	sErrorDescription1 := 'User High level error.  Illegal demand data was transmitted.';				
	sErrorDescription2 := 'Check program';				
					
9070:					
					
	sErrorDescription1 := 'User High level error.  Illegal demand data was transmitted.';				
	sErrorDescription2 := 'Check program';				
					
9071:					
					
	sErrorDescription1 := 'User High level error.  Illegal demand data was transmitted.';				
	sErrorDescription2 := 'Check program';				
					
9072:					
					
	sErrorDescription1 := 'User High level error.  Illegal demand data was transmitted.';				
	sErrorDescription2 := 'Check program';				
					
9073:					
					
	sErrorDescription1 := 'User High level error.  Illegal demand data was transmitted.';				
	sErrorDescription2 := 'Check program';				
					
9074:					
					
	sErrorDescription1 := 'User High level error.  Illegal demand data was transmitted.';				
	sErrorDescription2 := 'Check program';				
					
9075:					
					
	sErrorDescription1 := 'User High level error.  Illegal demand data was transmitted.';				
	sErrorDescription2 := 'Check program';				
					
9076:					
					
	sErrorDescription1 := 'User High level error.  Illegal demand data was transmitted.';				
	sErrorDescription2 := 'Check program';				
					
9077:					
					
	sErrorDescription1 := 'User High level error.  Illegal demand data was transmitted.';				
	sErrorDescription2 := 'Check program';				
					
9078:					
					
	sErrorDescription1 := 'User High level error.  Illegal demand data was transmitted.';				
	sErrorDescription2 := 'Check program';				
					
9079:					
					
	sErrorDescription1 := 'User High level error.  Illegal demand data was transmitted.';				
	sErrorDescription2 := 'Check program';				
					
9080:					
					
	sErrorDescription1 := 'User High level error.  Illegal demand data was transmitted.';				
	sErrorDescription2 := 'Check program';				
					
9081:					
					
	sErrorDescription1 := 'User High level error.  Illegal demand data was transmitted.';				
	sErrorDescription2 := 'Check program';				
					
9082:					
					
	sErrorDescription1 := 'User High level error.  Illegal demand data was transmitted.';				
	sErrorDescription2 := 'Check program';				
					
9083:					
					
	sErrorDescription1 := 'User High level error.  Illegal demand data was transmitted.';				
	sErrorDescription2 := 'Check program';				
					
9084:					
					
	sErrorDescription1 := 'User High level error.  Illegal demand data was transmitted.';				
	sErrorDescription2 := 'Check program';				
					
9085:					
					
	sErrorDescription1 := 'User High level error.  Illegal demand data was transmitted.';				
	sErrorDescription2 := 'Check program';				
					
9086:					
					
	sErrorDescription1 := 'User High level error.  Illegal demand data was transmitted.';				
	sErrorDescription2 := 'Check program';				
					
9087:					
					
	sErrorDescription1 := 'User High level error.  Illegal demand data was transmitted.';				
	sErrorDescription2 := 'Check program';				
					
9088:					
					
	sErrorDescription1 := 'User High level error.  Illegal demand data was transmitted.';				
	sErrorDescription2 := 'Check program';				
					
9089:					
					
	sErrorDescription1 := 'User High level error.  Illegal demand data was transmitted.';				
	sErrorDescription2 := 'Check program';				
					
9090:					
					
	sErrorDescription1 := 'User High level error.  Illegal demand data was transmitted.';				
	sErrorDescription2 := 'Check program';				
					
9091:					
					
	sErrorDescription1 := 'User High level error.  Illegal demand data was transmitted.';				
	sErrorDescription2 := 'Check program';				
					
9092:					
					
	sErrorDescription1 := 'User High level error.  Illegal demand data was transmitted.';				
	sErrorDescription2 := 'Check program';				
					
9093:					
					
	sErrorDescription1 := 'User High level error.  Illegal demand data was transmitted.';				
	sErrorDescription2 := 'Check program';				
					
9094:					
					
	sErrorDescription1 := 'User High level error.  Illegal demand data was transmitted.';				
	sErrorDescription2 := 'Check program';				
					
9095:					
					
	sErrorDescription1 := 'User High level error.  Illegal demand data was transmitted.';				
	sErrorDescription2 := 'Check program';				
					
9096:					
					
	sErrorDescription1 := 'User High level error.  Illegal demand data was transmitted.';				
	sErrorDescription2 := 'Check program';				
					
9097:					
					
	sErrorDescription1 := 'User High level error.  Illegal demand data was transmitted.';				
	sErrorDescription2 := 'Check program';				
					
9098:					
					
	sErrorDescription1 := 'User High level error.  Illegal demand data was transmitted.';				
	sErrorDescription2 := 'Check program';				
					
9099:					
					
	sErrorDescription1 := 'User High level error.  Illegal demand data was transmitted.';				
	sErrorDescription2 := 'Check program';				
		
		END_CASE
END_IF		
		
IF bErrorRCActive AND bLowLevelErrorRCActive  THEN
		
		CASE udiLowLevelErrorId OF
			

0030:	
	
	sErrorDescription1 := 'Hand error. LS release  Hand error signal is input';
	sErrorDescription2 := 'Restore with LS release operation';
	
0031:	
	
	sErrorDescription1 := 'Air pressure errorAir pressure error signal input';
	sErrorDescription2 := 'Check Air pressure';
	
0091:	
	
	sErrorDescription1 := 'Can not access the Special signThis signal cannot be used in duplicate';
	sErrorDescription2 := 'Change output No or special output assignment parameter';
	
0092:	
	
	sErrorDescription1 := ' Can not use Electric hand signaThe output signal for the electric hand cannot be used';
	sErrorDescription2 := 'Correct the program';
	
0095:	
	
	sErrorDescription1 := ' Brake release switch is turniCannot execute while brake release switch is turning on.';
	sErrorDescription2 := 'Please check the brake release switch and turn it off.';
	
0101:	
	
	sErrorDescription1 := 'Temperature in the Controlle FAN check or Filter at the bottom on Controller becomes old';
	sErrorDescription2 := 'Please exchange the filter to new filter or clean up the filter';
	
0104:	
	
	sErrorDescription1 := ' Temp. in robot CPU is too higAmbient temperature of robot CPU becomes high';
	sErrorDescription2 := 'Please lower ambient temperature to the specification range';
	
0110:	
	
	sErrorDescription1 := ' Overload(UPS)The UPS is spent';
	sErrorDescription2 := 'Replace the UPS';
	
0113:	
	
	sErrorDescription1 := ' UPS power supply error UPS power supply is out OF range';
	sErrorDescription2 := 'Check the UPS power supply';
	
0301:	
	
	sErrorDescription1 := ' CR800 test L-ErrorGeneral-purpose L-Error for the function test of CR800';
	sErrorDescription2 := 'Check the embedded message';
	
0480:	
	
	sErrorDescription1 := ' THR-RR error(Add.Axis)Overheating of the regenerative resistor (Add.Axis) was detected';
	sErrorDescription2 := 'Exchange the cooling fan of the regenerative resistor (Add.Axis)';
	
1640:	
	
	sErrorDescription1 := 'Cannot servo ON (DEADMAN OFF)The servo cannot be turned ON while the deadman switch OFF';
	sErrorDescription2 := 'Turn the deadman switch ON before turning the servo ON';
	
1820:	
	
	sErrorDescription1 := 'Pos. data disagree.Check origPosition data changed during power off';
	sErrorDescription2 := 'Check the origin, re-install if neccesary';
	
1830:	
	
	sErrorDescription1 := 'JRC. Exseeds the Pos. limitExceeds the pos. limit by JRC command';
	sErrorDescription2 := 'Check current pos. and limit';
	
1840:	
	
	sErrorDescription1 := 'JRC Qtt. Setting Too LargeExceeds the Limit of JRC Move Qtt.';
	sErrorDescription2 := 'Modify Parameter JRCQTT';
	
1860:	
	
	sErrorDescription1 := 'Illegal parameter (TLC)The setting of parameter TLC is illegal';
	sErrorDescription2 := 'Correct the parameter TLC (=X/Y/Z)';
	
1862:	
	
	sErrorDescription1 := 'Illegal parameter (Servo DataThe setting of parameter for Servo Data Log is illegal';
	sErrorDescription2 := 'Correct the parameter for Servo Data Log';
	
1863:	
	
	sErrorDescription1 := ' Illegal parameter (F.Ctrl)The setting of parameter for F.Ctrl, F.Test function is illegal';
	sErrorDescription2 := 'Correct the parameter for F.Ctrl, F.Test function';
	
1864:	
	
	sErrorDescription1 := ' Illegal parameter (FTP)The setting of parameter for FTP is illegal';
	sErrorDescription2 := 'Correct the parameter for FTP';
	
1865:	
	
	sErrorDescription1 := ' Illegal parameter (OADL)The setting of parameter for OADL is illegal';
	sErrorDescription2 := 'Make the parameter equal to or higher than 1 IT time';
	
1866:	
	
	sErrorDescription1 := ' Rotary axis existsTo include a rotary axis, multi axes AACC cannot be designated';
	sErrorDescription2 := 'Please designate single axis AACC';
	
2000:	
	
	sErrorDescription1 := 'The servo is OFFThe servo is OFF so the robot will not operate';
	sErrorDescription2 := 'Turn the servo ON and then restart';
	
2010:	
	
	sErrorDescription1 := 'Pulse output was not possibleThere is an error in the pulse output designation';
	sErrorDescription2 := 'Correct the robot program';
	
2020:	
	
	sErrorDescription1 := 'Reading external position datThe command cannot be executed while reading ext. position data';
	sErrorDescription2 := 'Correct the robot program';
	
2030:	
	
	sErrorDescription1 := 'JOG operation cannot be accepJOG operation request was issued when it could not be accepted';
	sErrorDescription2 := 'Request again';
	
2041:	
	
	sErrorDescription1 := ' Cal. error of frame conv. cooSame positions or 3 points line up straight';
	sErrorDescription2 := 'Please change the definition position of the coordinate';
	
2042:	
	
	sErrorDescription1 := ' Frame conv. coord. is not setFrame conv. is executed though the coordinate is not set';
	sErrorDescription2 := 'Please set coordinate or stop the execution of the frame conv.';
	
2050:	
	
	sErrorDescription1 := ' CPU processing time exceedsBecause the function made effective is many at the same time';
	sErrorDescription2 := 'Refer to manual (Troubleshooting)';
	
2270:	
	
	sErrorDescription1 := ' Cannot servo ON (SS1/STO actiThe servo cannot be turned ON while SS1/STO is active';
	sErrorDescription2 := 'Disable SS1 before turning the servo ON';
	
2400:	
	
	sErrorDescription1 := ' Collision avoidance detectA collision avoidance was detected';
	sErrorDescription2 := 'Release the collision avoidance state';
	
2410:	
	
	sErrorDescription1 := ' Collision avoidance detectA collision avoidance was detected';
	sErrorDescription2 := 'Release the collision avoidance state';
	
2421:	
	
	sErrorDescription1 := ' A lot of colli. avoidance modA lot of collision avoidance models';
	sErrorDescription2 := 'Reduce the collision avoidance models';
	
2430:	
	
	sErrorDescription1 := ' Collision avoidance re-detectCollision avoidance was already detected';
	sErrorDescription2 := 'Release the collision avoidance state';
	
2510:	
	
	sErrorDescription1 := 'Tracking parameter reversesTracking parameter[EXCRGM*] Setting value reverses';
	sErrorDescription2 := 'Check the parameter[EXCRGM*] value.';
	
2520:	
	
	sErrorDescription1 := 'Tracking parameter is range oTracking parameter[TRBUF] Setting value is range over';
	sErrorDescription2 := 'Check the parameter[TRUBF] value.';
	
2530:	
	
	sErrorDescription1 := 'There is no area where data iThere is no area where data is written.';
	sErrorDescription2 := 'Please read the data by using TRRD';
	
2540:	
	
	sErrorDescription1 := 'There is no read data.There is no read data. ';
	sErrorDescription2 := 'Please use TRRD after executing TRWRT.';
	
2560:	
	
	sErrorDescription1 := 'Ilegal parameter of TrackingIlegal parameter of Tracking.';
	sErrorDescription2 := 'Please check the value of parameter.';
	
2580:	
	
	sErrorDescription1 := ' Workpiece is not in tracking aWorkpiece of tracking target is not in tracking area';
	sErrorDescription2 := 'Execute TrkMv On when there is workpiece in tracking area';
	
2600:	
	
	sErrorDescription1 := ' Position data exceeds the limPosition data exceeds the limit';
	sErrorDescription2 := 'Change the position data';
	
2601:	
	
	sErrorDescription1 := 'Start pos. exseeds the limitStart position data exceeds the limit';
	sErrorDescription2 := 'Change the start position data';
	
2602:	
	
	sErrorDescription1 := 'DSTN pos. exseeds the limitDestination position data exceeds the limit';
	sErrorDescription2 := 'Change the position data';
	
2603:	
	
	sErrorDescription1 := 'Med pos. data exseeds the limIntermediate position data exceeds the limit';
	sErrorDescription2 := 'Change the position data';
	
2610:	
	
	sErrorDescription1 := ' Error concerning spline (fileThe error concerning the spline file occurred';
	sErrorDescription2 := 'Please confirm the content by a detailed number of the error Please confirm the file number and the existence of the file Please write it again after preserving the spline file again Please confirm the versions of spline file and controller
							Please execute it after the spline interpolation ends Please open the spline file';
	
2611:	
	
	sErrorDescription1 := ' Error concerning spline (pathThe error concerning the path point occurred';
	sErrorDescription2 := 'Please confirm the content by a detailed number of the error Please review the position of the path point or the speed
							Please reduce the posture change Please correct a posture flag of the path point to the same';
	
2612:	
	
	sErrorDescription1 := ' Error concerning spline (condThe error concerning the execution condition occurred';
	sErrorDescription2 := 'Please confirm the content by a detailed number of the error Please do not use the spline interpolation. Please do not use the spline interpolation with ALWAYS/ERROR
							Please do not execute two or more splines at the same time. Please do not execute the step return';
	
2613:	
	
	sErrorDescription1 := ' Error concerning spline (procThe error occurred in the processing of the spline interpolation';
	sErrorDescription2 := 'Please confirm the content by a detailed number of the error. Please increase an effective path point to four points or more. Please add the path point of circular arc
							Please confirm the content of the spline file. Please decrease the load to the program execution. Please confirm the content of the spline file and MvSpl';
	
2614:	
	
	sErrorDescription1 := ' Error concerning spline (combThe function cannot be used at the same time with the spline';
	sErrorDescription2 := 'Please confirm the content by a detailed number of the error. Please execute the spline when the tracking is invalid
							Please change after the spline interpolation ends. Please execute after the spline interpolation ends';
	
2615:	
	
	sErrorDescription1 := ' Error concerning spline (rangA set value outside range exists for the spline interpolation';
	sErrorDescription2 := 'Please confirm the content by a detailed number of the error. Please change to substitute the value within the range';
	
2621:	
	
	sErrorDescription1 := ' Tracking function is effectivTracking and Ex-T cannot be executed at the same time';
	sErrorDescription2 := 'Please execute Ex-T when the tracking is invalid';
	
2622:	
	
	sErrorDescription1 := ' Singular point function is efSingular point and Ex-T cannot be executed at the same time';
	sErrorDescription2 := 'Please execute Ex-T when the singular point function is invalid';
	
2660:	
	
	sErrorDescription1 := ' Error concerning axis coopThe error concerning the axis coop occurred';
	sErrorDescription2 := 'Please Confirm the content by a detail number of the error';
	
2661:	
	
	sErrorDescription1 := ' Error concerning axis coop (cThe function cannot be used at the same time with the axis coop';
	sErrorDescription2 := 'Please confirm the content by a detailed number of the error';
	
2662:	
	
	sErrorDescription1 := ' Work setting cannot be changeThe additional axis tracking is executing';
	sErrorDescription2 := 'Please change after the work coop is invalid';
	
2700:	
	
	sErrorDescription1 := 'CMP error (different mode)The designated mode is different from the current mode';
	sErrorDescription2 := 'Execute CMP OFF and then designate';
	
2750:	
	
	sErrorDescription1 := 'Cannot execute while trackingCannot execute while tracking';
	sErrorDescription2 := 'Execute TRK OFF and then execute';
	
2800:	
	
	sErrorDescription1 := 'Illegal position dataIllegal position data';
	sErrorDescription2 := 'Change the position data';
	
2801:	
	
	sErrorDescription1 := 'Illegal position data (start)Illegal position data (start)';
	sErrorDescription2 := 'Change the position data';
	
2802:	
	
	sErrorDescription1 := 'Illegal position data (dstn)Illegal position data (dstn)';
	sErrorDescription2 := 'Change the position data';
	
2803:	
	
	sErrorDescription1 := 'Illegal position data (intmedIllegal position data (intmed)';
	sErrorDescription2 := 'Change the position data';
	
2804:	
	
	sErrorDescription1 := 'SPDOPT can not be operatedA singular point area exists on the locus';
	sErrorDescription2 := 'Change a interpolation type or destination position';
	
2810:	
	
	sErrorDescription1 := 'Posture flag is disagreePosture flag is different between current and destination';
	sErrorDescription2 := 'Change the position data';
	
2830:	
	
	sErrorDescription1 := 'Illegal posture ipol typeIllegal posture ipol type';
	sErrorDescription2 := 'Please check the TYPE value';
	
2900:	
	
	sErrorDescription1 := 'System ERROR MO0An error occurred in the internal processing';
	sErrorDescription2 := 'Please call S.C.';
	
2910:	
	
	sErrorDescription1 := 'Cannot move.(Brake is Locked)Cannot move.(Brake is Locked)';
	sErrorDescription2 := 'Release the brake lock axis.';
	
3100:	
	
	sErrorDescription1 := 'PROC stack overThere is an error in the program';
	sErrorDescription2 := 'Correct the program and re-execute';
	
3110:	
	
	sErrorDescription1 := 'Argument value range overArgument value range over';
	sErrorDescription2 := 'Check the argument range and reinput';
	
3120:	
	
	sErrorDescription1 := 'No. of arguments is overNo. of argument is over';
	sErrorDescription2 := 'Check the No. of arguments and reinput';
	
3130:	
	
	sErrorDescription1 := 'COM file is already openedCOM file is already opened';
	sErrorDescription2 := 'Check the file No. and re-execute';
	
3140:	
	
	sErrorDescription1 := 'Can not open COM file. Can not open COM file';
	sErrorDescription2 := 'Check the file No. and re-execute';
	
3141:	
	
	sErrorDescription1 := ' The NVOPEN is not executedThe NVOPEN is not executed';
	sErrorDescription2 := 'Check the file No. and re-execute';
	
3142:	
	
	sErrorDescription1 := ' Can not open COM line.Can NOT open COM line';
	sErrorDescription2 := 'Check the COM No. and re-execute';
	
3143:	
	
	sErrorDescription1 := ' Command is not executedA necessary command is not executed';
	sErrorDescription2 := 'Check the file No. and re-execute';
	
3144:	
	
	sErrorDescription1 := ' The file dose not exist.The specified file does not exist.';
	sErrorDescription2 := 'Confirm the file name.';
	
3145:	
	
	sErrorDescription1 := ' The file cannot read.The learning file was broken.';
	sErrorDescription2 := 'Please learn again.';
	
3150:	
	
	sErrorDescription1 := 'Cannnot PTINT (INPUT mode)The file open mode is INPUT, so PRINT is not possible';
	sErrorDescription2 := 'Check the file No., open mode and re-execute';
	
3151:	
	
	sErrorDescription1 := 'A file with the same name exiA file with the same name already exists.';
	sErrorDescription2 := 'Confirm the file name.';
	
3170:	
	
	sErrorDescription1 := 'Cannot INPUT (OUTPUT mode)The file open mode is OUTPUT, so INPUT is not possible';
	sErrorDescription2 := 'Check the file No., open mode and re-execute';
	
3180:	
	
	sErrorDescription1 := 'System error (array range oveSystem error (array range over)';
	sErrorDescription2 := 'Please call S.C.';
	
3200:	
	
	sErrorDescription1 := 'This file is read onlyThis file is read only';
	sErrorDescription2 := 'Check the file';
	
3210:	
	
	sErrorDescription1 := 'This variable is write protecThis variable is write protected';
	sErrorDescription2 := 'Check the variable protection setting';
	
3220:	
	
	sErrorDescription1 := 'Nesting overNesting over';
	sErrorDescription2 := 'Correct the program and re-execute';
	
3230:	
	
	sErrorDescription1 := 'FOR NEXT statements unmatchFOR NEXT statements unmatch';
	sErrorDescription2 := 'Correct the program and re-execute';
	
3240:	
	
	sErrorDescription1 := ' Nesting over (FOR,WHILE)Nesting over (FOR,WHILE)';
	sErrorDescription2 := 'Correct the program and re-execute';
	
3250:	
	
	sErrorDescription1 := 'WHILE WEND statements unmatchWHILE WEND statements unmatch';
	sErrorDescription2 := 'Correct the program and re-execute';
	
3251:	
	
	sErrorDescription1 := 'Number of jump destination exNumber of jump destination exceeds 32';
	sErrorDescription2 := 'Correct the program and re-execute';
	
3252:	
	
	sErrorDescription1 := 'IF ENDIF statements unmatchIF ENDIF statements unmatch';
	sErrorDescription2 := 'Correct the program and re-execute';
	
3253:	
	
	sErrorDescription1 := 'Nesting over (IF,ENDIF)Nesting over (IF,ENDIF)';
	sErrorDescription2 := 'Correct the program and re-execute';
	
3254:	
	
	sErrorDescription1 := 'SELECT END SELECT statements SELECT END SELECT statements unmatch';
	sErrorDescription2 := 'Correct the program and re-execute';
	
3255:	
	
	sErrorDescription1 := 'IF ELSE statements unmatchIF ELSE statements unmatch';
	sErrorDescription2 := 'Correct the program and re-execute';
	
3256:	
	
	sErrorDescription1 := ' Function definition errorThe error concerning the function definition occurred. ';
	sErrorDescription2 := 'Please confirm the content by a detailed number of the error. ';
	
3257:	
	
	sErrorDescription1 := ' Include declaration errorThe error concerning the include declaration occurred.';
	sErrorDescription2 := 'Please confirm the content by a detailed number of the error. ';
	
3258:	
	
	sErrorDescription1 := ' Preprocessor errorThe error concerning the preprocessor occurred. ';
	sErrorDescription2 := 'Please confirm the content by a detailed number of the error. ';
	
3260:	
	
	sErrorDescription1 := 'Cannot exec for all slotsCannot exec for all slots';
	sErrorDescription2 := 'Exec for individual slot';
	
3262:	
	
	sErrorDescription1 := ' Illegal parameter setting HOEIllegal parameter setting HOE';
	sErrorDescription2 := 'Correct parameter HOE';
	
3270:	
	
	sErrorDescription1 := 'The command size is exceededThe command size is exceeded';
	sErrorDescription2 := 'Use 256 characters or less';
	
3280:	
	
	sErrorDescription1 := 'Cannot execute without GETMCannot execute without GETM';
	sErrorDescription2 := 'Execute the GETM command and then execute';
	
3281:	
	
	sErrorDescription1 := 'Cannot execute during RUNCannot execute during RUN';
	sErrorDescription2 := 'Cannot execute during RUN';
	
3282:	
	
	sErrorDescription1 := 'Can not RUN(not select, attribuThe program is not selected or the attribute is illegal';
	sErrorDescription2 := 'Select program or change the attribute';
	
3284:	
	
	sErrorDescription1 := ' Cannot execute while editingCannot execute while editing';
	sErrorDescription2 := 'Cannot execute while editing';
	
3285:	
	
	sErrorDescription1 := 'Cannot execute (RUN or WAI)Cannot execute (RUN or WAI)';
	sErrorDescription2 := 'Execute Program Reset';
	
3286:	
	
	sErrorDescription1 := 'Program is emptyProgram is empty';
	sErrorDescription2 := 'Edit program or select correct program';
	
3287:	
	
	sErrorDescription1 := 'Cannot execute (ERROR ALWAYS)The start condition is ERROR or ALWAYS';
	sErrorDescription2 := 'Correct the program';
	
3288:	
	
	sErrorDescription1 := 'Cannot execute while editingCannot execute while editing';
	sErrorDescription2 := 'Cannot execute while editing';
	
3289:	
	
	sErrorDescription1 := 'Program does not exist (SLT*)The program designated in the parameter SLT* does not exist';
	sErrorDescription2 := 'Correct parameter SLT*';
	
3290:	
	
	sErrorDescription1 := 'System slot cannot be executeSystem slot cannot be executed';
	sErrorDescription2 := 'Check whether another slot (user slot) is being operated';
	
3300:	
	
	sErrorDescription1 := 'User slot cannot be executedUser slot cannot be executed';
	sErrorDescription2 := 'Check whether another slot (system slot) is being operated';
	
3310:	
	
	sErrorDescription1 := 'Cannot execute XRUN (Runing)The slot is already running';
	sErrorDescription2 := 'Stop the slot then execute XRUN';
	
3320:	
	
	sErrorDescription1 := 'Cannnot execute XRUN (empty)The slot is not selected program';
	sErrorDescription2 := 'Set the argument(program name) or execute XLOAD';
	
3330:	
	
	sErrorDescription1 := 'Cannnot execute XSTP (empty)The slot is not selected program';
	sErrorDescription2 := 'Correct the program and re-execute';
	
3340:	
	
	sErrorDescription1 := 'Cannnot execute XRST (empty)The slot is not selected program';
	sErrorDescription2 := 'The state of the slot is WAI';
	
3350:	
	
	sErrorDescription1 := 'Cannnot execute XRST (RunningThe slot is already running';
	sErrorDescription2 := 'Stop the slot then execute XRST';
	
3360:	
	
	sErrorDescription1 := 'Cannnot execute XLOAD (not PSThe state of the slot is RUN or WAI';
	sErrorDescription2 := 'Execute XRST then execute XLOAD';
	
3361:	
	
	sErrorDescription1 := 'Can not load the program(SLT*Can not load the program(SLT*)';
	sErrorDescription2 := 'Correct parameter SLT* or program size check';
	
3370:	
	
	sErrorDescription1 := 'Cannnot execute XCLR (empty)The slot is not selected program';
	sErrorDescription2 := 'The state of the slot is RUN or WAI';
	
3380:	
	
	sErrorDescription1 := 'Cannnot execute XCLR (not PSAThe state of the slot is RUN or WAI';
	sErrorDescription2 := 'Execute XRST then execute XCLR';
	
3390:	
	
	sErrorDescription1 := 'Cannot use arc palletCannot use arc pallet';
	sErrorDescription2 := 'Change to another method';
	
3391:	
	
	sErrorDescription1 := 'Cannot use MVA2Cannot use MVA2';
	sErrorDescription2 := 'Change to another method';
	
3400:	
	
	sErrorDescription1 := 'System error (PROC stack overSystem error (PROC stack over)';
	sErrorDescription2 := 'Check System.When it comes back, contact to the dealer.';
	
3500:	
	
	sErrorDescription1 := 'Ilegal format input (INPUT)Ilegal format input (INPUT)';
	sErrorDescription2 := 'Check the format';
	
3501:	
	
	sErrorDescription1 := ' Illegal Receive data (EBREAD)Type is different (receive data and specified variable)';
	sErrorDescription2 := 'Please confirm specified tag data of the vision';
	
3502:	
	
	sErrorDescription1 := ' Illegal receive formatThe specified format is not corresponding to the received data';
	sErrorDescription2 := 'Check the content of the receive data';
	
3600:	
	
	sErrorDescription1 := 'Jump destination does not exiThe jump destination does not exist. Illegal execution line number.';
	sErrorDescription2 := 'Check the jump destination. Please operate it again after doing program reset.';
	
3601:	
	
	sErrorDescription1 := ' Jump destination is incorrectJumping into program control block is prohibited. ';
	sErrorDescription2 := 'Correct the program and re-execute. ';
	
3700:	
	
	sErrorDescription1 := 'Undefined variableUse of an undefined variable was attempted';
	sErrorDescription2 := 'Define the variable before using it';
	
3710:	
	
	sErrorDescription1 := 'Nesting over (CALLP)CALLP is used for seven or more stages';
	sErrorDescription2 := 'Check the program';
	
3720:	
	
	sErrorDescription1 := 'RC NX statements unmatchRC NX statements unmatch';
	sErrorDescription2 := 'Correct the program and re-execute';
	
3730:	
	
	sErrorDescription1 := ' Error of GETPOS statementError of GETPOS statement';
	sErrorDescription2 := 'Correct the program and re-execute';
	
3740:	
	
	sErrorDescription1 := ' There are a lot of BreakpointBreakpoint are up to 8';
	sErrorDescription2 := 'Please release an unnecessary breakpoint';
	
3750:	
	
	sErrorDescription1 := ' Illegal positions (DEF PLT)Multi rotation flag (FL2 J1/J2/J4 axis) is different';
	sErrorDescription2 := 'Specify positions to become the same multi rotation flag';
	
3760:	
	
	sErrorDescription1 := ' Illegal positions (DEF PLT)J1 or J4 axis is greatly changed (DEF PLT)';
	sErrorDescription2 := 'Specify positions to be not different greatly';
	
3770:	
	
	sErrorDescription1 := ' Undefined Mo-triggerUse of an undefined Mo-trigger was attempted';
	sErrorDescription2 := 'Please use it after defining a specified Mo-trigger';
	
3780:	
	
	sErrorDescription1 := ' Cannot use the MELFA Smart PlInvalid MELFA Smart Plus.';
	sErrorDescription2 := 'Check the MELFA Smart Plus card or parameter.';
	
3781:	
	
	sErrorDescription1 := ' Cannot use the MELFA Smart PlInvalid MELFA Smart Plus.';
	sErrorDescription2 := 'Check the MELFA Smart Plus card or parameter.';
	
3782:	
	
	sErrorDescription1 := ' There are MELFA Smart Plus CarMultiple MELFA Smart Plus cards are installed.';
	sErrorDescription2 := 'Turn off controller and pull unnecessary MELFA Smart Plus card.';
	
3800:	
	
	sErrorDescription1 := ' Cannot use this command.It is necessary to release the using permission.';
	sErrorDescription2 := 'Contact the maker';
	
3801:	
	
	sErrorDescription1 := ' Cannot execute this command.The usage of this command is incorrect.';
	sErrorDescription2 := 'Please check the specification of this command.';
	
3810:	
	
	sErrorDescription1 := 'Different argument typeThe argument type is different';
	sErrorDescription2 := 'Designate the correct argument';
	
3820:	
	
	sErrorDescription1 := 'Undefined intermediate codeThere is an error in the input syntax';
	sErrorDescription2 := 'Check the input syntax';
	
3821:	
	
	sErrorDescription1 := ' A compilation error occuredThere is an error in the input syntax. ';
	sErrorDescription2 := 'Check the error number in the error message. ';
	
3830:	
	
	sErrorDescription1 := 'Cannot execute GETMCannot execute GETM';
	sErrorDescription2 := 'Check whether the robot are being used with other slot';
	
3840:	
	
	sErrorDescription1 := 'RETURN without GOSUBRETURN was executed without using GOSUB';
	sErrorDescription2 := 'Check the program';
	
3850:	
	
	sErrorDescription1 := 'Undefined PLTAn undefined PLT is being used';
	sErrorDescription2 := 'Define PLT before using it';
	
3860:	
	
	sErrorDescription1 := 'Illegal position data definedThe definition of the position data is illegal';
	sErrorDescription2 := 'Check The definition of the position data';
	
3870:	
	
	sErrorDescription1 := 'Illegal mech No.The designated mech No. is an invalid value';
	sErrorDescription2 := 'Input the correct mech No';
	
3880:	
	
	sErrorDescription1 := 'Illegal slot No.The designated slot No. is an invalid value';
	sErrorDescription2 := 'Input the correct slot No';
	
3890:	
	
	sErrorDescription1 := 'System error (make MCODE)System error (make MCODE)';
	sErrorDescription2 := 'Correct to the backup-data';
	
3900:	
	
	sErrorDescription1 := 'JRC Command is disableCannot execute (JRC)';
	sErrorDescription2 := 'Cannot execute (JRC)';
	
3910:	
	
	sErrorDescription1 := 'Cannnot execute (JRC 0)The axis No is illegal (JRC)';
	sErrorDescription2 := 'Correctly set';
	
3920:	
	
	sErrorDescription1 := ' Palletize data errorCheck palletize data';
	sErrorDescription2 := 'Check palletize data';
	
3930:	
	
	sErrorDescription1 := ' This command cannot be executCollision detection is effective';
	sErrorDescription2 := 'Repeal collision detection (execute COLCHK OFF)';
	
3940:	
	
	sErrorDescription1 := 'COLCHK cannot be executedAn exclusive function is performing with COLCHK. CMP command is executed. TORQ command is executed.';
	sErrorDescription2 := 'Repeal the corresponding function. Repeal compliance mode (execute CMP OFF). Repeal torque restrictions (execute TORQ <Ax-No.>,100)';
	
3950:	
	
	sErrorDescription1 := 'NOERR cannot be executedInterruption using M_COLSTS is invalid';
	sErrorDescription2 := 'Define interruption using M_COLSTS and confirm it';
	
3960:	
	
	sErrorDescription1 := 'This ACT No. cannot be repealNOERR of collision detection is performed';
	sErrorDescription2 := 'Repeal this interruption after canceling NOERR';
	
3970:	
	
	sErrorDescription1 := 'COLCHK cannot be performedCollision detection serves as prohibition of use';
	sErrorDescription2 := 'Change parameter COL into use permission';
	
3980:	
	
	sErrorDescription1 := 'M_LDM cannot be executedPREC or MvTune command is executed';
	sErrorDescription2 := 'Repeal high accuracy mode (execute PREC OFF or MvTune 1)';
	
3981:	
	
	sErrorDescription1 := 'PREC cannot be executedM_LDM command is executed';
	sErrorDescription2 := 'Set load mode 1 (execute M_LDM=0)';
	
3982:	
	
	sErrorDescription1 := 'Cannot be used (singular poin This robot does not correspond to the singular point function. CMP command is executed. A synchronous addition axis control is effective Tracking mode is effective. Pre-fetch execution is effective. This robot is a setting of the multi mechan';
	sErrorDescription2 := 'Check the argument of TYPE specification. Invalidate a compliance mode (execute CMP OFF). Invalidate a synchronous addition axis control Invalidate a tracking mode (execute TRK OFF). Invalidate a pre-fetch execution';
	
3984:	
	
	sErrorDescription1 := 'Cannot be passsed (singularitRobot passes position which is very near the singular point';
	sErrorDescription2 := 'Adjust the teaching position';
	
3986:	
	
	sErrorDescription1 := ' Force control effective errorIt is an error concerning effective of the force control';
	sErrorDescription2 := 'Please confirm the setting';
	
3987:	
	
	sErrorDescription1 := ' F.Ctrl command execution erroIt is an error concerning the force control command execution';
	sErrorDescription2 := 'Please confirm the execution condition of the command';
	
3990:	
	
	sErrorDescription1 := 'COLCHK cannot be usedThis robot is a setting of the multi mechanism';
	sErrorDescription2 := 'Change parameter COL into use prohibition';
	
3991:	
	
	sErrorDescription1 := 'Mainte.Forecast cannot be useThis robot is a setting of the multi mechanism';
	sErrorDescription2 := 'Invalidate the maintenance forecast';
	
3994:	
	
	sErrorDescription1 := ' Can not use Shared Memory with CPU Shared Memory Function can not be used with MB4';
	sErrorDescription2 := 'Change RLNG parameter to 2(MB5)';
	
3995:	
	
	sErrorDescription1 := ' Can not use SQ Direct AND ALWEN. Can NOT use SQ Direct AND ALWENA';
	sErrorDescription2 := 'Change ALWENA parameter to 0';
	
3996:	
	
	sErrorDescription1 := ' Can not use SQ Direct with MB4SQ Direct Execution Function can not be used with MB4';
	sErrorDescription2 := 'Change RLNG parameter to 2(MB5)';
	
3998:	
	
	sErrorDescription1 := ' Parameter is wrong (OPNONE).OPNONE parameter setting is illegal.';
	sErrorDescription2 := 'Return OPNONE parameter to an initial value.';
	
3999:	
	
	sErrorDescription1 := ' Parameter is wrong (OPSIMPLE)OPSIMPLE parameter setting is illegal.';
	sErrorDescription2 := 'Return OPSIMPLE parameter to an initial value.';
	
4000:	
	
	sErrorDescription1 := 'System error (time out)System error (time out)';
	sErrorDescription2 := 'Check System.When it comes back, contact to the dealer.';
	
4100:	
	
	sErrorDescription1 := 'No. of registered file is fulThe number of registered file has been exceeded';
	sErrorDescription2 := 'Delete any unnecessary programs';
	
4110:	
	
	sErrorDescription1 := 'Memory area is fullMemory area is full';
	sErrorDescription2 := 'Delete any unnecessary programs or data';
	
4120:	
	
	sErrorDescription1 := 'Too long program nameThe program name is a maximum of 12 characters';
	sErrorDescription2 := 'Set the program name to within 12 characters';
	
4130:	
	
	sErrorDescription1 := 'Illegal program nameAn illegal character was used in the program name';
	sErrorDescription2 := 'Only numbers and alphabetic characters can be used';
	
4140:	
	
	sErrorDescription1 := 'The program was not foundThe designated program was not found';
	sErrorDescription2 := 'Designate a different program, or create the designated program';
	
4150:	
	
	sErrorDescription1 := 'Program is faultyProgram is faulty';
	sErrorDescription2 := 'Delete the program';
	
4160:	
	
	sErrorDescription1 := 'Not a robot programThe designated program is not a robot program';
	sErrorDescription2 := 'Designate a different program';
	
4170:	
	
	sErrorDescription1 := 'The program is being editedThe program is being edited';
	sErrorDescription2 := 'Close the program being edited';
	
4180:	
	
	sErrorDescription1 := 'Program is runningThe program is running';
	sErrorDescription2 := 'Stop the program';
	
4190:	
	
	sErrorDescription1 := 'The program is selectedThe program is selected';
	sErrorDescription2 := 'Execute program reset';
	
4200:	
	
	sErrorDescription1 := 'Cannot write to file1: Write protected, or 2: File capacity is too low';
	sErrorDescription2 := '1. Enable file writing, or 2: Delete unnecessary files';
	
4201:	
	
	sErrorDescription1 := ' Can not operate in ROM mode. Can not operate in ROM mode';
	sErrorDescription2 := 'Change to RAM mode';
	
4202:	
	
	sErrorDescription1 := ' Cannot read from fileRead protected';
	sErrorDescription2 := 'Enable file reading';
	
4210:	
	
	sErrorDescription1 := 'Too long statementThe command statement length is limited to 127 characters';
	sErrorDescription2 := 'Delete characters in the statement to within 127 characters';
	
4220:	
	
	sErrorDescription1 := 'Syntax errorThere is an error in the syntax of the input command statement';
	sErrorDescription2 := 'Check the program, and reinput the correct syntax';
	
4230:	
	
	sErrorDescription1 := 'The line No. does not existThe designated line No. does not exist';
	sErrorDescription2 := 'Check the program, and reinput the correct line No';
	
4240:	
	
	sErrorDescription1 := 'The statement is write protecThe command statement is write protected';
	sErrorDescription2 := 'Cancel the write protection';
	
4250:	
	
	sErrorDescription1 := 'No more lines or variablesReading of lines and variables exceeding the registered ones';
	sErrorDescription2 := 'Check the programs';
	
4300:	
	
	sErrorDescription1 := 'Too longvariable nameThe variable name length is limited to 8 characters';
	sErrorDescription2 := 'Shorten the variable name to within 8 characters';
	
4310:	
	
	sErrorDescription1 := 'Ilegal character is usedA character other than A to Z or 0 to 9 is used';
	sErrorDescription2 := 'Do not use illegal characters';
	
4320:	
	
	sErrorDescription1 := 'The variable is write protectThe variable is write protected';
	sErrorDescription2 := '1. Use a writable variable, or 2. Cancel the write protection';
	
4330:	
	
	sErrorDescription1 := 'The variable is read protecteThe variable is read protected';
	sErrorDescription2 := '1. Use a readable variable, or 2. Cancel the read protection';
	
4340:	
	
	sErrorDescription1 := 'The variable is not definedThe variable has not been defined';
	sErrorDescription2 := 'Define the variable';
	
4341:	
	
	sErrorDescription1 := ' The variable is not definedThe user external variable has not been defined';
	sErrorDescription2 := 'Define the user external variable';
	
4350:	
	
	sErrorDescription1 := 'Duplicate definition (Val.)Variables already defined cannot be redefined with DIM or DEF';
	sErrorDescription2 := '1. Change the name and define, or 2. Delete the variable';
	
4360:	
	
	sErrorDescription1 := 'Same variable used (65535 timThe same variable cannot be used more than 65535 times';
	sErrorDescription2 := 'Change program to reduce the times the same variable is used';
	
4370:	
	
	sErrorDescription1 := 'Error in the array element1.The elements exceeds the range, 2.The variable is not an array';
	sErrorDescription2 := '1. Correct the array element, or 2. Do not use an array element';
	
4380:	
	
	sErrorDescription1 := 'Cannot delete variables (usedVariables used in a command statement cannot be deleted';
	sErrorDescription2 := 'Delete the command statement using the variable';
	
4390:	
	
	sErrorDescription1 := 'Variable type combination errThe user-defined global variable type differs in LOCAL and BASE';
	sErrorDescription2 := 'Match the variable types';
	
4400:	
	
	sErrorDescription1 := 'Program is faulty.Program is faulty';
	sErrorDescription2 := 'Delete the program';
	
4410:	
	
	sErrorDescription1 := 'Renumbering data errorRenumbering data error';
	sErrorDescription2 := 'Check the program and reset the data';
	
4420:	
	
	sErrorDescription1 := 'Line No exceeds 32767The new line No. or line gap is large';
	sErrorDescription2 := 'Do not use line Nos. exceeding 32767';
	
4430:	
	
	sErrorDescription1 := 'Not found the string searchedThe character string searched for was not found';
	sErrorDescription2 := 'Check the program';
	
4440:	
	
	sErrorDescription1 := 'Duplicate definition (label)A label already defined cannot be redefined';
	sErrorDescription2 := '1. Change the label name, or 2. Delete the defined label line';
	
4450:	
	
	sErrorDescription1 := 'The variable No. is out of raPosition/counter/string No. is out of range';
	sErrorDescription2 := 'Change the variable No. into the correct range';
	
4460:	
	
	sErrorDescription1 := 'Argument value range overArgument value range over';
	sErrorDescription2 := 'Check the argument range and reinput';
	
4470:	
	
	sErrorDescription1 := 'Line No can not be usedLine No can not be used';
	sErrorDescription2 := 'Please use the label';
	
4800:	
	
	sErrorDescription1 := 'System error (System base proThe system base program name is not correctly set';
	sErrorDescription2 := 'Correctly set the system base program in the parameter';
	
4810:	
	
	sErrorDescription1 := 'The global variable defined bThe parameter "PRGUSR" is not correctly set';
	sErrorDescription2 := 'Correctly set the user base program in the parameter PRGUSR';
	
4811:	
	
	sErrorDescription1 := 'The global variable redefinedA system global variable is defined in user global';
	sErrorDescription2 := 'Correct the program';
	
4820:	
	
	sErrorDescription1 := 'No editing programThe editing program has been closed';
	sErrorDescription2 := 'Try editing the program again';
	
4900:	
	
	sErrorDescription1 := 'System error (Prog Hndl)The program name used by internal processing is not normal.';
	sErrorDescription2 := 'Check System.When it comes back, contact to the dealer.';
	
4910:	
	
	sErrorDescription1 := 'Robot Language is mismatchedThe parameter RLNG is mismatched';
	sErrorDescription2 := 'Correct RLNG or select another program';
	
4920:	
	
	sErrorDescription1 := 'There is no backup data in ROThere is no backup data in ROM';
	sErrorDescription2 := 'Please operate after backup';
	
4921:	
	
	sErrorDescription1 := ' Not support this robot languaIllegal robot language setting.';
	sErrorDescription2 := 'Please confirm the language setting.';
	
4922:	
	
	sErrorDescription1 := ' Unsupported program versionThis program was created with the new version. ';
	sErrorDescription2 := 'This program cannot be opened with this robot. ';
	
4930:	
	
	sErrorDescription1 := ' CAVCHK cannot be executedThe collision avoidance is set at unusable';
	sErrorDescription2 := 'Change parameter CAV into usable';
	
4931:	
	
	sErrorDescription1 := ' CMP command cannot be executeCollision avoidance is effective';
	sErrorDescription2 := 'Invalidate collision avoidance (execute CAVCHK OFF)';
	
4932:	
	
	sErrorDescription1 := ' TRK command cannot be executeCollision avoidance is effective';
	sErrorDescription2 := 'Invalidate collision avoidance (execute CAVCHK OFF)';
	
4933:	
	
	sErrorDescription1 := ' CavChk cannot be executed (CMCMP command is executed';
	sErrorDescription2 := 'Invalidate compliance mode (execute CMP OFF)';
	
4934:	
	
	sErrorDescription1 := ' CavChk cannot be executed (TRTRK command is executed';
	sErrorDescription2 := 'Invalidate tracking mode (execute TRK OFF)';
	
4935:	
	
	sErrorDescription1 := ' NOERR cannot be executedInterruption using M_CAVSTS is invalid';
	sErrorDescription2 := 'Define interruption using M_CAVSTS and confirm it';
	
4936:	
	
	sErrorDescription1 := ' This ACT No. cannot be repealNOERR of collision avoidance is performed';
	sErrorDescription2 := 'Repeal this interruption after canceling NOERR';
	
4937:	
	
	sErrorDescription1 := ' A user free area size is lackThe size of a user free area is smaller than that of 2K';
	sErrorDescription2 := 'Please set 2K or more to the size of a user free area';
	
4938:	
	
	sErrorDescription1 := ' This robot does not corresponThis robot does not correspond to collision avoidance';
	sErrorDescription2 := 'Parameter CAV returns disapproval';
	
4939:	
	
	sErrorDescription1 := ' CAV version of other CPU is oSoftware version of other CPU is old';
	sErrorDescription2 := 'Contact the maker';
	
4941:	
	
	sErrorDescription1 := ' MvSpl command cannot be execuCollision avoidance is effective';
	sErrorDescription2 := 'Invalidate collision avoidance (execute CAVCHK OFF)';
	
4950:	
	
	sErrorDescription1 := ' Error in a function syntaxError in the definition of a function procedure. ';
	sErrorDescription2 := 'Correct the definition of the function procedure. ';
	
5010:	
	
	sErrorDescription1 := 'AUTOENA signal is OFFAUTOENA  signal is OFF';
	sErrorDescription2 := 'ON the AUTOENA signal, or enter the TEACH mode';
	
5100:	
	
	sErrorDescription1 := 'No program is selectedA program is not selected for the designated slot';
	sErrorDescription2 := 'Select a program for the designated slot';
	
5110:	
	
	sErrorDescription1 := 'Continuous RUN is not possiblA different program name has been designated';
	sErrorDescription2 := 'Designate the correct program name';
	
5120:	
	
	sErrorDescription1 := 'Cannot select program (not PSThe designated slot is not in the program selection state';
	sErrorDescription2 := 'Reset the program';
	
5130:	
	
	sErrorDescription1 := 'Cannot execute servo onA servo OFF process is taking place';
	sErrorDescription2 := 'Wait for the servo to turn OFF before turning the servo ON';
	
5140:	
	
	sErrorDescription1 := 'Cannot read the fileNow reading or it is already editting';
	sErrorDescription2 := 'Close the file or retry after';
	
5150:	
	
	sErrorDescription1 := 'The origin has not been setThe origin has not been set';
	sErrorDescription2 := 'Set the origin';
	
5200:	
	
	sErrorDescription1 := 'Parameter error (TASKMAX)The No. of multi tasks has exceeded the limit';
	sErrorDescription2 := 'Reduce the No. of multi tasks';
	
5210:	
	
	sErrorDescription1 := 'Parameter error (MECHAMAX)The No. of multi robot has exceeded the limit';
	sErrorDescription2 := 'Reduce the No. of multi robot';
	
5400:	
	
	sErrorDescription1 := 'All robot cannot be designateAll robot cannot be designated';
	sErrorDescription2 := 'Designate an independent robot No';
	
5410:	
	
	sErrorDescription1 := 'Non-existent modeNon-existent mode was designated';
	sErrorDescription2 := 'Designate the correct mode';
	
5420:	
	
	sErrorDescription1 := 'Illegal slot No.The slot No. designation is illegal';
	sErrorDescription2 := 'Designate the correct slot No.';
	
5430:	
	
	sErrorDescription1 := 'Illegal robot No.The robot No. designation is illegal';
	sErrorDescription2 := 'Designate the correct robot No.';
	
5600:	
	
	sErrorDescription1 := 'Cannot execute during an erroCannot execute during an error';
	sErrorDescription2 := 'Reset the error';
	
5620:	
	
	sErrorDescription1 := 'Cannot execute during CSTOP OCannot execute during cycle stop signal input';
	sErrorDescription2 := 'Turn the cycle stop signal OFF';
	
5630:	
	
	sErrorDescription1 := 'Cannot execute during SRVOFF Cannot execute during servo OFF signal input';
	sErrorDescription2 := 'Turn the SRVOFF signal OFF';
	
5640:	
	
	sErrorDescription1 := 'Cannot execute during RUNCannot execute during RUN';
	sErrorDescription2 := 'Stop  and then execute';
	
5650:	
	
	sErrorDescription1 := 'Cannot execute during STOPCannot execute during stop';
	sErrorDescription2 := 'Complete the stop, and then execute';
	
5660:	
	
	sErrorDescription1 := 'Edit during RUN(include ALWAYEdit during RUN(include ALWAYS)';
	sErrorDescription2 := 'Complete the stop, and then execute';
	
5990:	
	
	sErrorDescription1 := 'System error (Illegal commandNot exist command was executed.';
	sErrorDescription2 := 'Designate the correct command';
	
6010:	
	
	sErrorDescription1 := 'Illegal commandA non-registered command was sent';
	sErrorDescription2 := 'Input the correct command';
	
6011:	
	
	sErrorDescription1 := ' Cannot connect to CR800Cannot connect to CR800';
	sErrorDescription2 := 'Please connect to CPU unit';
	
6020:	
	
	sErrorDescription1 := 'The Operation is disableThe Operation is disable';
	sErrorDescription2 := 'Acquire the operation enable';
	
6030:	
	
	sErrorDescription1 := 'The editing operation is disaThe editing operation is disable';
	sErrorDescription2 := 'Acquire the editing operation enable';
	
6040:	
	
	sErrorDescription1 := 'System error (illegal device A non-registered device No. was set.';
	sErrorDescription2 := 'Designate the correct device';
	
6130:	
	
	sErrorDescription1 := ' Network Communication errorNetwork fail or Parameter setting is illegal';
	sErrorDescription2 := 'Please check the network cable or parameter';
	
6190:	
	
	sErrorDescription1 := ' Network error generationNetwork error occurred';
	sErrorDescription2 := 'Please confirm the content of the network error';
	
6600:	
	
	sErrorDescription1 := 'COMDEV parameter is illegalUndefined signal number';
	sErrorDescription2 := 'Set the correct signal number';
	
6610:	
	
	sErrorDescription1 := 'Cannot output (hand input)The hand input signal cannot be written';
	sErrorDescription2 := 'Use an output signal';
	
6620:	
	
	sErrorDescription1 := 'Cannot write (special INPUT)Cannot write (special INPUT)';
	sErrorDescription2 := 'Use an real signal mode';
	
6630:	
	
	sErrorDescription1 := 'Input signal cannot be writteThis is the actual signal input mode';
	sErrorDescription2 := 'Set a pseudo-input signal mode';
	
6631:	
	
	sErrorDescription1 := ' Input Skip signal cannot be wThis is the actual signal input mode';
	sErrorDescription2 := 'Use an real signal mode';
	
6632:	
	
	sErrorDescription1 := ' Input TREN signal cannot be wThis is the actual signal input mode';
	sErrorDescription2 := 'Use an real signal mode';
	
6641:	
	
	sErrorDescription1 := 'Duplicate setting (special INThe special input signal has been defined in duplicate';
	sErrorDescription2 := 'Correct the parameter';
	
6642:	
	
	sErrorDescription1 := 'STOP is fixed signal No.The parameter cannot be changed';
	sErrorDescription2 := 'The parameter STOP(input) return to an initial value';
	
6643:	
	
	sErrorDescription1 := 'Illegal parameter (special SiThe parameter setting is illegal';
	sErrorDescription2 := 'Set the bigger No to the start No than the end No';
	
6650:	
	
	sErrorDescription1 := 'Duplicate setting (special OUThe Special output signal has been defined in duplicate';
	sErrorDescription2 := 'Correct the parameter';
	
6651:	
	
	sErrorDescription1 := 'Duplicate setting (HANDTYPE)The Special output signal has been defined in duplicate';
	sErrorDescription2 := 'Correct the parameter';
	
6660:	
	
	sErrorDescription1 := 'Cannot output (SPECIAL OUT)The program setting is illegal';
	sErrorDescription2 := 'Correct the program';
	
6670:	
	
	sErrorDescription1 := 'Illegal OUT reset patternThe parameters are not defined in sets of 8 characters';
	sErrorDescription2 := 'Check the parameter ORST0,..,ORST224';
	
6800:	
	
	sErrorDescription1 := 'Cancel pseudo-input mode, PW The pseudo-input mode was canceled';
	sErrorDescription2 := 'Turn the power OFF';
	
6990:	
	
	sErrorDescription1 := ' Illegal user macro signal inpTwo or more user macro input signals are input at the same time.';
	sErrorDescription2 := 'Please input the user macro input signal individually.';
	
7071:	
	
	sErrorDescription1 := 'Not enough memory area for CTContinue function needs more than 100Kbytes memory area';
	sErrorDescription2 := 'Delete unnecessary programs';
	
7072:	
	
	sErrorDescription1 := 'Memory area is fullMemory area is full';
	sErrorDescription2 := 'Delete any unnecessary programs or data';
	
7099:	
	
	sErrorDescription1 := ' Can not read parameter[%s]The parameter does not exist';
	sErrorDescription2 := 'Please confirm the parameter';
	
7301:	
	
	sErrorDescription1 := ' Parameter was changedA new set value is not reflected in the robot controller';
	sErrorDescription2 := 'Turn the power OFF and ON once';
	
7311:	
	
	sErrorDescription1 := 'The power was OFF during filePower off during file saving';
	sErrorDescription2 := 'Please do not carry out power off during file saving';
	
7330:	
	
	sErrorDescription1 := ' Can not change in ROM mode.Can not change in ROM mode';
	sErrorDescription2 := 'Please change to RAM mode and perform again';
	
7331:	
	
	sErrorDescription1 := ' Can not change memory size in R Can not change memory size in ROM mode';
	sErrorDescription2 := 'Please change to RAM mode and perform again';
	
7332:	
	
	sErrorDescription1 := 'Can not change to RAM mode in C Can not change to ROM mode in continue mode';
	sErrorDescription2 := 'Please change to RAM mode and perform again';
	
7340:	
	
	sErrorDescription1 := 'Contine function cannot be usContine function cannot be used in DRAM mode';
	sErrorDescription2 := 'Please change to RAM mode and perform again';
	
7341:	
	
	sErrorDescription1 := 'Can not change to DRAM mode in Can not change to DRAM mode in CTN mode';
	sErrorDescription2 := 'Please change to RAM mode and perform again';
	
7342:	
	
	sErrorDescription1 := 'Global extension cannot be usGlobal extension cannot be used in DRAM mode';
	sErrorDescription2 := 'Please change to RAM mode and perform again';
	
7343:	
	
	sErrorDescription1 := 'Can not change to DRAM mode in Can not change to DRAM mode in PRGGBL mode';
	sErrorDescription2 := 'Please change to RAM mode and perform again';
	
7370:	
	
	sErrorDescription1 := ' The password is 8 to 32 char.The password is 8 to 32 characters';
	sErrorDescription2 := 'Please input the password 8 to 32 characters';
	
7371:	
	
	sErrorDescription1 := 'Only alphanumeric characterIt input it excluding the alphanumeric character';
	sErrorDescription2 := 'Please input the password in the alphanumeric character';
	
7372:	
	
	sErrorDescription1 := ' The password is unmatchThe password is unmatch';
	sErrorDescription2 := 'Please input the password again';
	
7373:	
	
	sErrorDescription1 := ' Password lock to the programsPassword lock to the programs';
	sErrorDescription2 := 'Please release password';
	
7374:	
	
	sErrorDescription1 := ' Password lock to the parametePassword lock to the parameter';
	sErrorDescription2 := 'Please release password';
	
7375:	
	
	sErrorDescription1 := ' Password lock to the filesPassword lock to the files';
	sErrorDescription2 := 'Please release password';
	
7376:	
	
	sErrorDescription1 := ' The password is 1000 to 99999The password is 1000 to 999999999';
	sErrorDescription2 := 'Please input the password 1000 to 999999999';
	
7377:	
	
	sErrorDescription1 := ' Password lock to the programPassword lock to the program';
	sErrorDescription2 := 'Please release password';
	
7378:	
	
	sErrorDescription1 := ' Change the passwordThe password has not been changed from an initial value';
	sErrorDescription2 := 'Please change to a new password';
	
7400:	
	
	sErrorDescription1 := ' Form of backup file is differThis file is for the maintenance forecast of other methods';
	sErrorDescription2 := 'Please select the backup file for a present method';
	
7680:	
	
	sErrorDescription1 := ' Test processing errorThe error occurred when the test processing was executed';
	sErrorDescription2 := 'Please confirm the test method';
	
7730:	
	
	sErrorDescription1 := ' CC-Link Data link errorIllegal communication line or change the master parameter';
	sErrorDescription2 := 'Check the cable or master parameters';
	
7750:	
	
	sErrorDescription1 := ' CC-Link Master Parameter erroIllegal communication line or illegal master parameter setting';
	sErrorDescription2 := 'Check the cable or master parameters';
	
7780:	
	
	sErrorDescription1 := ' Illegal CC-Link register numbIllegal CC-Link register number';
	sErrorDescription2 := 'Input the correct number';
	
7781:	
	
	sErrorDescription1 := ' INPUT signal No. is for CC-LiINPUT signal No. is for CC-Link';
	sErrorDescription2 := 'Install CC-Link card';
	
7850:	
	
	sErrorDescription1 := ' Cannot read MXT positional daThe format of MXT positional data file is illegal.';
	sErrorDescription2 := 'Please confirm the format of a positional data file. ';
	
7940:	
	
	sErrorDescription1 := ' Solder cont. communication erSolder controller communication error';
	sErrorDescription2 := 'Check the connection solder controller, communication setting';
	
7941:	
	
	sErrorDescription1 := ' Solder cont. range overSolder controller range over';
	sErrorDescription2 := 'Please confirm a set value of the solder controller';
	
8050:	
	
	sErrorDescription1 := ' ';
	sErrorDescription2 := '';
	
8051:	
	
	sErrorDescription1 := ' ';
	sErrorDescription2 := '';
	
8052:	
	
	sErrorDescription1 := ' ';
	sErrorDescription2 := '';
	
8053:	
	
	sErrorDescription1 := ' ';
	sErrorDescription2 := '';
	
8054:	
	
	sErrorDescription1 := ' ';
	sErrorDescription2 := '';
	
8055:	
	
	sErrorDescription1 := ' ';
	sErrorDescription2 := '';
	
8056:	
	
	sErrorDescription1 := ' ';
	sErrorDescription2 := '';
	
8057:	
	
	sErrorDescription1 := ' ';
	sErrorDescription2 := '';
	
8059:	
	
	sErrorDescription1 := ' ';
	sErrorDescription2 := '';
	
8060:	
	
	sErrorDescription1 := ' ';
	sErrorDescription2 := '';
	
8061:	
	
	sErrorDescription1 := ' ';
	sErrorDescription2 := '';
	
8062:	
	
	sErrorDescription1 := ' ';
	sErrorDescription2 := '';
	
8063:	
	
	sErrorDescription1 := ' ';
	sErrorDescription2 := '';
	
8064:	
	
	sErrorDescription1 := ' ';
	sErrorDescription2 := '';
	
8065:	
	
	sErrorDescription1 := ' ';
	sErrorDescription2 := '';
	
8066:	
	
	sErrorDescription1 := ' ';
	sErrorDescription2 := '';
	
8067:	
	
	sErrorDescription1 := ' ';
	sErrorDescription2 := '';
	
8068:	
	
	sErrorDescription1 := ' ';
	sErrorDescription2 := '';
	
8069:	
	
	sErrorDescription1 := ' ';
	sErrorDescription2 := '';
	
8070:	
	
	sErrorDescription1 := ' ';
	sErrorDescription2 := '';
	
8071:	
	
	sErrorDescription1 := ' ';
	sErrorDescription2 := '';
	
8072:	
	
	sErrorDescription1 := ' ';
	sErrorDescription2 := '';
	
8073:	
	
	sErrorDescription1 := ' ';
	sErrorDescription2 := '';
	
8074:	
	
	sErrorDescription1 := ' ';
	sErrorDescription2 := '';
	
8075:	
	
	sErrorDescription1 := ' ';
	sErrorDescription2 := '';
	
8076:	
	
	sErrorDescription1 := ' ';
	sErrorDescription2 := '';
	
8077:	
	
	sErrorDescription1 := ' ';
	sErrorDescription2 := '';
	
8078:	
	
	sErrorDescription1 := ' ';
	sErrorDescription2 := '';
	
8079:	
	
	sErrorDescription1 := ' ';
	sErrorDescription2 := '';
	
8090:	
	
	sErrorDescription1 := ' ';
	sErrorDescription2 := '';
	
8100:	
	
	sErrorDescription1 := ' ';
	sErrorDescription2 := '';
	
8101:	
	
	sErrorDescription1 := ' ';
	sErrorDescription2 := '';
	
8102:	
	
	sErrorDescription1 := ' ';
	sErrorDescription2 := '';
	
8103:	
	
	sErrorDescription1 := ' ';
	sErrorDescription2 := '';
	
8104:	
	
	sErrorDescription1 := ' ';
	sErrorDescription2 := '';
	
8105:	
	
	sErrorDescription1 := ' ';
	sErrorDescription2 := '';
	
8106:	
	
	sErrorDescription1 := ' ';
	sErrorDescription2 := '';
	
8107:	
	
	sErrorDescription1 := ' ';
	sErrorDescription2 := '';
	
8108:	
	
	sErrorDescription1 := ' ';
	sErrorDescription2 := '';
	
8109:	
	
	sErrorDescription1 := ' ';
	sErrorDescription2 := '';
	
8110:	
	
	sErrorDescription1 := ' ';
	sErrorDescription2 := '';
	
8111:	
	
	sErrorDescription1 := ' ';
	sErrorDescription2 := '';
	
8141:	
	
	sErrorDescription1 := ' Electric hand1 Alarm occurAlarm of Electric hand was detected';
	sErrorDescription2 := 'Please remove cause of alarm referring to electric hand manual';
	
8142:	
	
	sErrorDescription1 := ' Electric hand1 Error occurError of Electric hand was detected';
	sErrorDescription2 := 'Please remove cause of error referring to electric hand manual';
	
8143:	
	
	sErrorDescription1 := ' Electric hand1 UnconnectionElectric hand is not connected';
	sErrorDescription2 := 'Check the communication cable connection and Station No. setting';
	
8144:	
	
	sErrorDescription1 := ' Electric hand1 type is not seType selection of Electric hand is not completed';
	sErrorDescription2 := 'Please select the type of Electric hand by parameter setting';
	
8145:	
	
	sErrorDescription1 := ' Electric hand1 origin is not Original position return of Electric hand is not completed';
	sErrorDescription2 := 'Please execute original position return';
	
8146:	
	
	sErrorDescription1 := ' Electric hand1 Response timeoCable connection is bad,or electric hand breakdown';
	sErrorDescription2 := 'Confirm cable connection and hand state, and the power OFF';
	
8147:	
	
	sErrorDescription1 := ' Electric hand1 Command doubleElectric hand operation command was doubly executed';
	sErrorDescription2 := 'Please correct the program,or review the operating procedure';
	
8148:	
	
	sErrorDescription1 := ' Electric hand1 Point setting The registration of the electric hand point data overlapped';
	sErrorDescription2 := 'Please correct the program,or review the operating procedure';
	
8149:	
	
	sErrorDescription1 := ' Electric hand1 system fault3The system fault occurred in electric hand';
	sErrorDescription2 := 'After reset error, please execute original position return';
	
8151:	
	
	sErrorDescription1 := ' Electric hand2 Alarm occurAlarm of Electric hand was detected';
	sErrorDescription2 := 'Please remove cause of alarm referring to electric hand manual';
	
8152:	
	
	sErrorDescription1 := ' Electric hand2 Error occurError of Electric hand was detected';
	sErrorDescription2 := 'Please remove cause of error referring to electric hand manual';
	
8153:	
	
	sErrorDescription1 := ' Electric hand2 UnconnectionElectric hand is not connected';
	sErrorDescription2 := 'Check the communication cable connection and Station No. setting';
	
8154:	
	
	sErrorDescription1 := ' Electric hand2 type is not seType selection of Electric hand is not completed';
	sErrorDescription2 := 'Please select the type of Electric hand by parameter setting';
	
8155:	
	
	sErrorDescription1 := ' Electric hand2 origin is not Original position return of Electric hand is not completed';
	sErrorDescription2 := 'Please execute original position return';
	
8156:	
	
	sErrorDescription1 := ' Electric hand2 Response timeoCable connection is bad,or electric hand breakdown';
	sErrorDescription2 := 'Confirm cable connection and hand state, and the power OFF';
	
8157:	
	
	sErrorDescription1 := ' Electric hand2 Command doubleElectric hand operation command was doubly executed';
	sErrorDescription2 := 'Please correct the program,or review the operating procedure';
	
8158:	
	
	sErrorDescription1 := ' Electric hand2 Point setting The registration of the electric hand point data overlapped';
	sErrorDescription2 := 'Please correct the program,or review the operating procedure';
	
8159:	
	
	sErrorDescription1 := ' Electric hand2 system fault3The system fault occurred in electric hand';
	sErrorDescription2 := 'After reset error, please execute original position return';
	
8161:	
	
	sErrorDescription1 := ' Electric hand3 Alarm occurAlarm of Electric hand was detected';
	sErrorDescription2 := 'Please remove cause of alarm referring to electric hand manual';
	
8162:	
	
	sErrorDescription1 := ' Electric hand3 Error occurError of Electric hand was detected';
	sErrorDescription2 := 'Please remove cause of error referring to electric hand manual';
	
8163:	
	
	sErrorDescription1 := ' Electric hand3 UnconnectionElectric hand is not connected';
	sErrorDescription2 := 'Check the communication cable connection and Station No. setting';
	
8164:	
	
	sErrorDescription1 := ' Electric hand3 type is not seType selection of Electric hand is not completed';
	sErrorDescription2 := 'Please select the type of Electric hand by parameter setting';
	
8165:	
	
	sErrorDescription1 := ' Electric hand3 origin is not Original position return of Electric hand is not completed';
	sErrorDescription2 := 'Please execute original position return';
	
8166:	
	
	sErrorDescription1 := ' Electric hand3 Response timeoCable connection is bad,or electric hand breakdown';
	sErrorDescription2 := 'Confirm cable connection and hand state, and the power OFF';
	
8167:	
	
	sErrorDescription1 := ' Electric hand3 Command doubleElectric hand operation command was doubly executed';
	sErrorDescription2 := 'Please correct the program,or review the operating procedure';
	
8168:	
	
	sErrorDescription1 := ' Electric hand3 Point setting The registration of the electric hand point data overlapped';
	sErrorDescription2 := 'Please correct the program,or review the operating procedure';
	
8169:	
	
	sErrorDescription1 := ' Electric hand3 system fault3The system fault occurred in electric hand';
	sErrorDescription2 := 'After reset error, please execute original position return';
	
8300:	
	
	sErrorDescription1 := 'There are a lot of GETPOS defGETPOS function are up to 8';
	sErrorDescription2 := 'Please use the same ACT No. or reset an unnecessary program';
	
8310:	
	
	sErrorDescription1 := 'GETPOS undefinedGETPOS undefined';
	sErrorDescription2 := 'Please define GETPOS';
	
8330:	
	
	sErrorDescription1 := ' The watch condition is abnormThe watch condition cannot be changed (DEF GPS/MAP)';
	sErrorDescription2 := 'Please change the watch condition after executing GPSCHK OFF';
	
8331:	
	
	sErrorDescription1 := ' Duplicate definition (DEF GPSThe watch number is used by other slots (DEF GPS/MAP)';
	sErrorDescription2 := 'Please change to the watch number not used by another slot';
	
8430:	
	
	sErrorDescription1 := ' DEVICENET communication errorNetwork fail or Master setting is illegal';
	sErrorDescription2 := 'Please confirm network (speed,cable,terminator) or master unit';
	
8440:	
	
	sErrorDescription1 := ' DEVICENET Unit number overlapThere are more than one unit with same unit number on network';
	sErrorDescription2 := 'Please confirm the other unit number.';
	
8441:	
	
	sErrorDescription1 := ' DEVICENET Network power failuNetwork power is turned off.';
	sErrorDescription2 := 'Please turn on network power';
	
8442:	
	
	sErrorDescription1 := ' DEVICENET Other units not fouOther units are not connected on the network';
	sErrorDescription2 := 'Please confirm the other units';
	
8460:	
	
	sErrorDescription1 := ' DEVICENET timeoutDEVICENET timeout';
	sErrorDescription2 := 'Please confirm the other units or power supply of network';
	
8590:	
	
	sErrorDescription1 := ' FieldBUS card is not installeThe signal No. is for FieldBUS.';
	sErrorDescription2 := 'Install FieldBUS card.';
	
8600:	
	
	sErrorDescription1 := 'The vision is a unconnectionThe vision is a unconnection';
	sErrorDescription2 := 'Please check COM No. and Parameter';
	
8601:	
	
	sErrorDescription1 := 'The vision can not be logged onThe parameter of the user-name or the password is abnormal';
	sErrorDescription2 := 'Please set the parameter correctly';
	
8602:	
	
	sErrorDescription1 := 'Password is abnormalThe password of the user-name is not corresponding';
	sErrorDescription2 := 'Please set the password correctly';
	
8603:	
	
	sErrorDescription1 := 'Parameter is abnormalThe parameter of the user-name or the password is abnormal';
	sErrorDescription2 := 'Please set the parameter correctly';
	
8610:	
	
	sErrorDescription1 := 'The communication is abnormalThe communication was cut';
	sErrorDescription2 := 'Please check the communications cable';
	
8620:	
	
	sErrorDescription1 := 'The vision number is abnormalThe number is not designated by NVOPEN';
	sErrorDescription2 := 'Please check NVOPEN command';
	
8621:	
	
	sErrorDescription1 := 'Vision program name is abnormThe vision program name has exceeded 15 characters';
	sErrorDescription2 := 'Please make the program name within 15 characters';
	
8622:	
	
	sErrorDescription1 := 'There is no vision programThere is no specified vision program';
	sErrorDescription2 := 'Please check the vision program name';
	
8623:	
	
	sErrorDescription1 := ' SKIP number is already usedSKIP number is already used';
	sErrorDescription2 := 'Please confirm the SKIP number';
	
8630:	
	
	sErrorDescription1 := 'The recognition cell is illegThere is no value on the cell';
	sErrorDescription2 := 'Please check the recognition cell';
	
8631:	
	
	sErrorDescription1 := 'The cell is outside the rangeThe range of the cell is exceeded';
	sErrorDescription2 := 'Please check the range of the cell';
	
8632:	
	
	sErrorDescription1 := 'The vision is a time-outThere is no response from the vision';
	sErrorDescription2 := 'Please check the time-out time';
	
8633:	
	
	sErrorDescription1 := 'The vision is a time-out(NVTRThere is no response from the vision(NVTRG)';
	sErrorDescription2 := 'Please decrease the load of the network';
	
8634:	
	
	sErrorDescription1 := 'There is a comma within the rThere is a comma within the range of the cell';
	sErrorDescription2 := 'Please check the range of the cell';
	
8635:	
	
	sErrorDescription1 := 'There is no comma within the There is no comma within the range of the cell';
	sErrorDescription2 := 'Please check the range of the cell';
	
8636:	
	
	sErrorDescription1 := ' Vision Tag name abnormalThere is no specified vision tag in the vision program';
	sErrorDescription2 := 'Please correct the vision tag name';
	
8637:	
	
	sErrorDescription1 := ' Failure in writing data(EBWriSpecified tag name, data type, or value is illegal';
	sErrorDescription2 := 'Please check the tag name, the data type, and the value';
	
8640:	
	
	sErrorDescription1 := 'The image trigger is abnormalThe trigger setting of the vision sensor is abnormal';
	sErrorDescription2 := 'Please check the trigger setting';
	
8650:	
	
	sErrorDescription1 := 'Please make the vision onlineThe vision sensor is off-line';
	sErrorDescription2 := 'Please make vision sensor online';
	
8660:	
	
	sErrorDescription1 := 'There is no authorityThe authority of the user-name is not a full access';
	sErrorDescription2 := 'Please check user name';
	
8670:	
	
	sErrorDescription1 := 'Can not restartIt started without resetting it';
	sErrorDescription2 := 'Please reset the program';
	
8680:	
	
	sErrorDescription1 := ' Unknown code was receivedStatus code of unregistration was received from vision sensor';
	sErrorDescription2 := 'Please check communication state, setting, and command argument';
	
8690:	
	
	sErrorDescription1 := ' Vision communication errorThe communication error code returned from the vision sensor';
	sErrorDescription2 := 'Please refer to the manual of the vision sensor';
	
8700:	
	
	sErrorDescription1 := 'Multi CPU system self-check eIllegal parameter of multi CPU system and CPU is abnormal,etc. ';
	sErrorDescription2 := 'Confirm details and measures of the error with GX Developer etc.';
	
8710:	
	
	sErrorDescription1 := ' PC I/O module parameter%s errAn illegal setting of the PC I/O module was detected';
	sErrorDescription2 := 'Please check the value of parameter';
	
8720:	
	
	sErrorDescription1 := ' Fuse is blown.(PC I/O module)Fuse is blown.(PC I/O module)';
	sErrorDescription2 := 'Please refer to the manual of PC I/O module';
	
8730:	
	
	sErrorDescription1 := ' I/O module remove errorPC I/O module was removed';
	sErrorDescription2 := 'Please mount PC I/O module';
	
8881:	
	
	sErrorDescription1 := ' Transient processing errorThe demand data was transmitted while executing the transient';
	sErrorDescription2 := 'Please transmit after present processing ends';
	
8882:	
	
	sErrorDescription1 := ' Servo test unexecutionThe test of the servo testing function is not executed';
	sErrorDescription2 := 'Please execute the test of the servo testing function';
	
8883:	
	
	sErrorDescription1 := ' Servo test is incompleteThe test of the servo testing function is not completed';
	sErrorDescription2 := 'Please execute it after completing the test';
	
8884:	
	
	sErrorDescription1 := ' Command number range overThe command no. of the servo testing func. is outside the range';
	sErrorDescription2 := 'Please confirm the range and set a correct value';
	
8910:	
	
	sErrorDescription1 := ' Function uncorrespondenceThis robot cannot use this function';
	sErrorDescription2 := 'Do not use this function';
	
8911:	
	
	sErrorDescription1 := ' Set value is range overIt comes off from the range where a set value can be input';
	sErrorDescription2 := 'Change to the value which can be input';
	
8912:	
	
	sErrorDescription1 := ' Cannot repeat any furtherNecessary identification processing was completed';
	sErrorDescription2 := 'Check the frequency repeatedly';
	
8913:	
	
	sErrorDescription1 := ' All axes do not moveAn axis necessary for identification does not operate';
	sErrorDescription2 := 'Check a starting point and a destination in the program';
	
8914:	
	
	sErrorDescription1 := ' Execution order is wrongThe execution order is wrong';
	sErrorDescription2 := 'Check the execution order';
	
8915:	
	
	sErrorDescription1 := ' Data number shortageThe data used for identification is insufficient';
	sErrorDescription2 := 'Check the program. Especially, amount of movement and speed';
	
8916:	
	
	sErrorDescription1 := ' Identification operation erroIt became an error because of the identification processing';
	sErrorDescription2 := 'Check the program. Especially, amount of movement and speed';
	
8917:	
	
	sErrorDescription1 := ' The memory cannot be allocateA memory necessary for processing was not able to be allocated';
	sErrorDescription2 := 'Decrease the gathered volume of data';
	
8930:	
	
	sErrorDescription1 := ' Cannot be used (load estimatiThis robot does not correspond to the hand data estimation';
	sErrorDescription2 := 'Measure data directly from actual hand or workpiece';
	
9100:	
	
	sErrorDescription1 := ' User Low level errorIllegal demand data was transmitted';
	sErrorDescription2 := 'Check program';
	
9101:	
	
	sErrorDescription1 := ' User Low level errorIllegal demand data was transmitted';
	sErrorDescription2 := 'Check program';
	
9102:	
	
	sErrorDescription1 := ' User Low level errorIllegal demand data was transmitted';
	sErrorDescription2 := 'Check program';
	
9103:	
	
	sErrorDescription1 := 'User Low level errorIllegal demand data was transmitted';
	sErrorDescription2 := 'Check program';
	
9104:	
	
	sErrorDescription1 := 'User Low level errorIllegal demand data was transmitted';
	sErrorDescription2 := 'Check program';
	
9105:	
	
	sErrorDescription1 := 'User Low level errorIllegal demand data was transmitted';
	sErrorDescription2 := 'Check program';
	
9106:	
	
	sErrorDescription1 := 'User Low level errorIllegal demand data was transmitted';
	sErrorDescription2 := 'Check program';
	
9107:	
	
	sErrorDescription1 := 'User Low level errorIllegal demand data was transmitted';
	sErrorDescription2 := 'Check program';
	
9108:	
	
	sErrorDescription1 := 'User Low level errorIllegal demand data was transmitted';
	sErrorDescription2 := 'Check program';
	
9109:	
	
	sErrorDescription1 := 'User Low level errorIllegal demand data was transmitted';
	sErrorDescription2 := 'Check program';
	
9110:	
	
	sErrorDescription1 := ' User Low level errorIllegal demand data was transmitted';
	sErrorDescription2 := 'Check program';
	
9111:	
	
	sErrorDescription1 := ' User Low level errorIllegal demand data was transmitted';
	sErrorDescription2 := 'Check program';
	
9112:	
	
	sErrorDescription1 := ' User Low level errorIllegal demand data was transmitted';
	sErrorDescription2 := 'Check program';
	
9113:	
	
	sErrorDescription1 := ' User Low level errorIllegal demand data was transmitted';
	sErrorDescription2 := 'Check program';
	
9114:	
	
	sErrorDescription1 := ' User Low level errorIllegal demand data was transmitted';
	sErrorDescription2 := 'Check program';
	
9115:	
	
	sErrorDescription1 := ' User Low level errorIllegal demand data was transmitted';
	sErrorDescription2 := 'Check program';
	
9116:	
	
	sErrorDescription1 := ' User Low level errorIllegal demand data was transmitted';
	sErrorDescription2 := 'Check program';
	
9117:	
	
	sErrorDescription1 := 'User Low level errorIllegal demand data was transmitted';
	sErrorDescription2 := 'Check program';
	
9118:	
	
	sErrorDescription1 := 'User Low level errorIllegal demand data was transmitted';
	sErrorDescription2 := 'Check program';
	
9119:	
	
	sErrorDescription1 := 'User Low level errorIllegal demand data was transmitted';
	sErrorDescription2 := 'Check program';
	
9120:	
	
	sErrorDescription1 := ' User Low level errorIllegal demand data was transmitted';
	sErrorDescription2 := 'Check program';
	
9121:	
	
	sErrorDescription1 := ' User Low level errorIllegal demand data was transmitted';
	sErrorDescription2 := 'Check program';
	
9122:	
	
	sErrorDescription1 := ' User Low level errorIllegal demand data was transmitted';
	sErrorDescription2 := 'Check program';
	
9123:	
	
	sErrorDescription1 := ' User Low level errorIllegal demand data was transmitted';
	sErrorDescription2 := 'Check program';
	
9124:	
	
	sErrorDescription1 := 'User Low level errorIllegal demand data was transmitted';
	sErrorDescription2 := 'Check program';
	
9125:	
	
	sErrorDescription1 := 'User Low level errorIllegal demand data was transmitted';
	sErrorDescription2 := 'Check program';
	
9126:	
	
	sErrorDescription1 := 'User Low level errorIllegal demand data was transmitted';
	sErrorDescription2 := 'Check program';
	
9127:	
	
	sErrorDescription1 := 'User Low level errorIllegal demand data was transmitted';
	sErrorDescription2 := 'Check program';
	
9128:	
	
	sErrorDescription1 := 'User Low level errorIllegal demand data was transmitted';
	sErrorDescription2 := 'Check program';
	
9129:	
	
	sErrorDescription1 := 'User Low level errorIllegal demand data was transmitted';
	sErrorDescription2 := 'Check program';
	
9130:	
	
	sErrorDescription1 := 'User Low level errorIllegal demand data was transmitted';
	sErrorDescription2 := 'Check program';
	
9131:	
	
	sErrorDescription1 := 'User Low level errorIllegal demand data was transmitted';
	sErrorDescription2 := 'Check program';
	
9132:	
	
	sErrorDescription1 := 'User Low level errorIllegal demand data was transmitted';
	sErrorDescription2 := 'Check program';
	
9133:	
	
	sErrorDescription1 := 'User Low level errorIllegal demand data was transmitted';
	sErrorDescription2 := 'Check program';
	
9134:	
	
	sErrorDescription1 := 'User Low level errorIllegal demand data was transmitted';
	sErrorDescription2 := 'Check program';
	
9135:	
	
	sErrorDescription1 := 'User Low level errorIllegal demand data was transmitted';
	sErrorDescription2 := 'Check program';
	
9136:	
	
	sErrorDescription1 := 'User Low level errorIllegal demand data was transmitted';
	sErrorDescription2 := 'Check program';
	
9137:	
	
	sErrorDescription1 := 'User Low level errorIllegal demand data was transmitted';
	sErrorDescription2 := 'Check program';
	
9138:	
	
	sErrorDescription1 := 'User Low level errorIllegal demand data was transmitted';
	sErrorDescription2 := 'Check program';
	
9139:	
	
	sErrorDescription1 := 'User Low level errorIllegal demand data was transmitted';
	sErrorDescription2 := 'Check program';
	
9140:	
	
	sErrorDescription1 := 'User Low level errorIllegal demand data was transmitted';
	sErrorDescription2 := 'Check program';
	
9141:	
	
	sErrorDescription1 := 'User Low level errorIllegal demand data was transmitted';
	sErrorDescription2 := 'Check program';
	
9142:	
	
	sErrorDescription1 := 'User Low level errorIllegal demand data was transmitted';
	sErrorDescription2 := 'Check program';
	
9143:	
	
	sErrorDescription1 := 'User Low level errorIllegal demand data was transmitted';
	sErrorDescription2 := 'Check program';
	
9144:	
	
	sErrorDescription1 := 'User Low level errorIllegal demand data was transmitted';
	sErrorDescription2 := 'Check program';
	
9145:	
	
	sErrorDescription1 := 'User Low level errorIllegal demand data was transmitted';
	sErrorDescription2 := 'Check program';
	
9146:	
	
	sErrorDescription1 := 'User Low level errorIllegal demand data was transmitted';
	sErrorDescription2 := 'Check program';
	
9147:	
	
	sErrorDescription1 := 'User Low level errorIllegal demand data was transmitted';
	sErrorDescription2 := 'Check program';
	
9148:	
	
	sErrorDescription1 := 'User Low level errorIllegal demand data was transmitted';
	sErrorDescription2 := 'Check program';
	
9149:	
	
	sErrorDescription1 := 'User Low level errorIllegal demand data was transmitted';
	sErrorDescription2 := 'Check program';
	
9150:	
	
	sErrorDescription1 := 'User Low level errorIllegal demand data was transmitted';
	sErrorDescription2 := 'Check program';
	
9151:	
	
	sErrorDescription1 := 'User Low level errorIllegal demand data was transmitted';
	sErrorDescription2 := 'Check program';
	
9152:	
	
	sErrorDescription1 := 'User Low level errorIllegal demand data was transmitted';
	sErrorDescription2 := 'Check program';
	
9153:	
	
	sErrorDescription1 := 'User Low level errorIllegal demand data was transmitted';
	sErrorDescription2 := 'Check program';
	
9154:	
	
	sErrorDescription1 := 'User Low level errorIllegal demand data was transmitted';
	sErrorDescription2 := 'Check program';
	
9155:	
	
	sErrorDescription1 := 'User Low level errorIllegal demand data was transmitted';
	sErrorDescription2 := 'Check program';
	
9156:	
	
	sErrorDescription1 := 'User Low level errorIllegal demand data was transmitted';
	sErrorDescription2 := 'Check program';
	
9157:	
	
	sErrorDescription1 := 'User Low level errorIllegal demand data was transmitted';
	sErrorDescription2 := 'Check program';
	
9158:	
	
	sErrorDescription1 := 'User Low level errorIllegal demand data was transmitted';
	sErrorDescription2 := 'Check program';
	
9159:	
	
	sErrorDescription1 := 'User Low level errorIllegal demand data was transmitted';
	sErrorDescription2 := 'Check program';
	
9160:	
	
	sErrorDescription1 := 'User Low level errorIllegal demand data was transmitted';
	sErrorDescription2 := 'Check program';
	
9161:	
	
	sErrorDescription1 := 'User Low level errorIllegal demand data was transmitted';
	sErrorDescription2 := 'Check program';
	
9162:	
	
	sErrorDescription1 := 'User Low level errorIllegal demand data was transmitted';
	sErrorDescription2 := 'Check program';
	
9163:	
	
	sErrorDescription1 := 'User Low level errorIllegal demand data was transmitted';
	sErrorDescription2 := 'Check program';
	
9164:	
	
	sErrorDescription1 := 'User Low level errorIllegal demand data was transmitted';
	sErrorDescription2 := 'Check program';
	
9165:	
	
	sErrorDescription1 := 'User Low level errorIllegal demand data was transmitted';
	sErrorDescription2 := 'Check program';
	
9166:	
	
	sErrorDescription1 := 'User Low level errorIllegal demand data was transmitted';
	sErrorDescription2 := 'Check program';
	
9167:	
	
	sErrorDescription1 := 'User Low level errorIllegal demand data was transmitted';
	sErrorDescription2 := 'Check program';
	
9168:	
	
	sErrorDescription1 := 'User Low level errorIllegal demand data was transmitted';
	sErrorDescription2 := 'Check program';
	
9169:	
	
	sErrorDescription1 := 'User Low level errorIllegal demand data was transmitted';
	sErrorDescription2 := 'Check program';
	
9170:	
	
	sErrorDescription1 := ' User Low level errorIllegal demand data was transmitted';
	sErrorDescription2 := 'Check program';
	
9171:	
	
	sErrorDescription1 := ' User Low level errorIllegal demand data was transmitted';
	sErrorDescription2 := 'Check program';
	
9172:	
	
	sErrorDescription1 := 'User Low level errorIllegal demand data was transmitted';
	sErrorDescription2 := 'Check program';
	
9173:	
	
	sErrorDescription1 := 'User Low level errorIllegal demand data was transmitted';
	sErrorDescription2 := 'Check program';
	
9174:	
	
	sErrorDescription1 := 'User Low level errorIllegal demand data was transmitted';
	sErrorDescription2 := 'Check program';
	
9175:	
	
	sErrorDescription1 := 'User Low level errorIllegal demand data was transmitted';
	sErrorDescription2 := 'Check program';
	
9176:	
	
	sErrorDescription1 := 'User Low level errorIllegal demand data was transmitted';
	sErrorDescription2 := 'Check program';
	
9177:	
	
	sErrorDescription1 := 'User Low level errorIllegal demand data was transmitted';
	sErrorDescription2 := 'Check program';
	
9178:	
	
	sErrorDescription1 := 'User Low level errorIllegal demand data was transmitted';
	sErrorDescription2 := 'Check program';
	
9179:	
	
	sErrorDescription1 := 'User Low level errorIllegal demand data was transmitted';
	sErrorDescription2 := 'Check program';
	
9180:	
	
	sErrorDescription1 := 'User Low level errorIllegal demand data was transmitted';
	sErrorDescription2 := 'Check program';
	
9181:	
	
	sErrorDescription1 := ' User Low level errorIllegal demand data was transmitted';
	sErrorDescription2 := 'Check program';
	
9182:	
	
	sErrorDescription1 := ' User Low level errorIllegal demand data was transmitted';
	sErrorDescription2 := 'Check program';
	
9183:	
	
	sErrorDescription1 := ' User Low level errorIllegal demand data was transmitted';
	sErrorDescription2 := 'Check program';
	
9184:	
	
	sErrorDescription1 := ' User Low level errorIllegal demand data was transmitted';
	sErrorDescription2 := 'Check program';
	
9185:	
	
	sErrorDescription1 := 'User Low level errorIllegal demand data was transmitted';
	sErrorDescription2 := 'Check program';
	
9186:	
	
	sErrorDescription1 := 'User Low level errorIllegal demand data was transmitted';
	sErrorDescription2 := 'Check program';
	
9187:	
	
	sErrorDescription1 := 'User Low level errorIllegal demand data was transmitted';
	sErrorDescription2 := 'Check program';
	
9188:	
	
	sErrorDescription1 := 'User Low level errorIllegal demand data was transmitted';
	sErrorDescription2 := 'Check program';
	
9189:	
	
	sErrorDescription1 := 'User Low level errorIllegal demand data was transmitted';
	sErrorDescription2 := 'Check program';
	
9190:	
	
	sErrorDescription1 := 'User Low level errorIllegal demand data was transmitted';
	sErrorDescription2 := 'Check program';
	
9191:	
	
	sErrorDescription1 := ' User Low level errorIllegal demand data was transmitted';
	sErrorDescription2 := 'Check program';
	
9192:	
	
	sErrorDescription1 := ' User Low level errorIllegal demand data was transmitted';
	sErrorDescription2 := 'Check program';
	
9193:	
	
	sErrorDescription1 := ' User Low level errorIllegal demand data was transmitted';
	sErrorDescription2 := 'Check program';
	
9194:	
	
	sErrorDescription1 := ' User Low level errorIllegal demand data was transmitted';
	sErrorDescription2 := 'Check program';
	
9195:	
	
	sErrorDescription1 := 'User Low level errorIllegal demand data was transmitted';
	sErrorDescription2 := 'Check program';
	
9196:	
	
	sErrorDescription1 := 'User Low level errorIllegal demand data was transmitted';
	sErrorDescription2 := 'Check program';
	
9197:	
	
	sErrorDescription1 := 'User Low level errorIllegal demand data was transmitted';
	sErrorDescription2 := 'Check program';
	
9198:	
	
	sErrorDescription1 := 'User Low level errorIllegal demand data was transmitted';
	sErrorDescription2 := 'Check program';
	
9199:	
	
	sErrorDescription1 := 'User Low level errorIllegal demand data was transmitted';
	sErrorDescription2 := 'Check program';




		END_CASE
END_IF
sErrorDescription1 :=CONCAT(sErrorDescription1,': ');
sErrorDescription1 :=CONCAT(sErrorDescription1,sErrorDescription2);
END_ACTION

ACTION ErrorHandling:
//Alarm_0500	500	Error	Błąd robota {0}
IF bAlarmInit THEN
    bAlarmInit := FALSE; 
	fbSourceInfo.Clear();
	fbSourceInfo.sName:=sStationName;//'Machine';
	fbSourceInfo.nId:=iStationIndex;//2700;
	// Alarm_0500	500	Error	Błąd robota {0}
    arfbAlarm[0].CreateEx(stEventEntry := TC_EVENTS.AlarmClass.Alarm_0500, bWithConfirmation:= FALSE,  ipSourceInfo:= fbSourceInfo); 
END_IF


// Opźnienie na odczytanie kodu błędu z robota
tonbStateError(IN:= (eState = E_Station.eError) OR (eState = E_Station.eResetting), PT:=T#20MS);
bStateError	:=	tonbStateError.Q;

//tonErrorDelay(IN:=bErrorRCActive, PT:=T#200MS);
(*
IF eState = E_Station.eResetting THEN
	
	bResetErrorRC					:= bReset;
	eRunningState					:= E_RobotMovState.eReadyPlace;
	bHomingDone						:= FALSE;
	udiErrorId						:= 0;
	
ELSE
*)
(*	
	//IF tonErrorDelay.Q THEN
		bError						:= bErrorRCActive AND bEnable;
	//END_IF	
	
	IF bErrorRCActive THEN
		
		eState 						:= E_Station.eError;
		bErrorNumberRequest			:= TRUE;
		nErrorNr					:= IODATA;
		
	END_IF
	
	bResetErrorRC					:= FALSE;
	
	IF bEStop AND nErrorNr = 50 THEN
		bResetErrorRC				:= TRUE;
		//bHomingDone					:= FALSE;
	END_IF	
	
	CASE nErrorNr OF
		
		0001: sErrorDescription			:= 'Fail safe error (SRVOFF)';
		0002: sErrorDescription			:= 'Fail safe error (STOP)';
		0003: sErrorDescription			:= 'The system is abnormal.';	
		0004: sErrorDescription			:= 'CPU Watch dog error';	
		0039: sErrorDescription			:= 'Door Switch Signal line is faulty.';	
		0040: sErrorDescription			:= 'Door Switch Signal is Input';
		0041: sErrorDescription			:= 'Comm. error (Remote I/O #1).';
		0042: sErrorDescription			:= 'Comm. error (Remote I/O #2).';
		0044: sErrorDescription			:= 'OP Mode key line is faulty';
		0045: sErrorDescription			:= 'Faulty Line (T/B Enable Switch).';
		0046: sErrorDescription			:= 'Faulty wiring (Enabling Device).';
		0050: sErrorDescription			:= 'EMG signal is input. (external)';	
		0051: sErrorDescription			:= 'Wiring of the external emergency stop is abnormal.';	
		0084: sErrorDescription			:= 'Fuse is broken (O/P)';	
		0086: sErrorDescription			:= 'Hand module overcurrent';	
		0087: sErrorDescription			:= 'Fuse is blown.(Brake';	
		0088: sErrorDescription			:= 'Service I/F fuse error';	
		0090: sErrorDescription			:= 'DC24V fuse is blown';
		0091: sErrorDescription			:= 'Cant access the Special signal';
		0093: sErrorDescription			:= 'Safety relay fuse is blown';
		0094: sErrorDescription			:= 'The overcurrent in the T/B line.';
		0095: sErrorDescription			:= 'Brake release switch is turning on';
		0101: sErrorDescription			:= 'Temperature in the Controller is too high';
		0102: sErrorDescription			:= 'Temperature in the Controller is too high';
		0120: sErrorDescription			:= 'Instantaneous power failure';
		0130: sErrorDescription			:= 'The initialization connection error of system remote I/O.';
		0131: sErrorDescription			:= 'Plural Ope-panel are installed.';
		0140: sErrorDescription			:= 'Fuse is blown.(Safety unit)';
		0141: sErrorDescription			:= 'Wiring error of EMGIN connector.';
		0431: sErrorDescription			:= 'Servo amplifier motor overheat';
		0432: sErrorDescription			:= 'Servo amplifier motor overheat';
		0433: sErrorDescription			:= 'Servo amplifier motor overheat';	
		0434: sErrorDescription			:= 'Servo amplifier motor overheat';		
		1011: sErrorDescription			:= 'Wykrycie kolizji';
		1012: sErrorDescription			:= 'Wykrycie kolizji';
		1013: sErrorDescription			:= 'Wykrycie kolizji';
		1014: sErrorDescription			:= 'Wykrycie kolizji';
		
	END_CASE
	
*)
IF (bEnable) THEN
	IF  arfbAlarm[0].bActive AND bReset THEN
		bServoONRC			:= FALSE;
		bResetErrorRC		:=TRUE;
		arfbAlarm[0].Clear(nTimeStamp:=0, bResetConfirmation:= FALSE);
 	END_IF	
	IF bErrorRCActive AND (bHighLevelErrorRCActive OR bLowLevelErrorRCActive) (*AND NOT bStateError*)  THEN
		bServoONRC			:= FALSE;
// 		arfbAlarm[0].ipArguments.Clear() .AddUDInt(udiHeightServoErrorNr);
// 		IF NOT arfbAlarm[0].bActive THEN	
// 			arfbAlarm[0].Raise(nTimeStamp:=0);
// 		END_IF
// 	ELSE	
// 		IF  arfbAlarm[0].bActive AND bReset THEN
// 			arfbAlarm[0].Clear(nTimeStamp:=0, bResetConfirmation:= FALSE);
// 		END_IF
		IF NOT arfbAlarm[0].bActive THEN
			bErrorNumberRequest										:= TRUE;
		END_IF
	
		IF IODATA <> 50 AND bErrorNumberRequestActive  THEN	
			
				//bError											:= TRUE;
			IF bHighLevelErrorRCActive THEN
				udiHighLevelErrorId								:= IODATA;
				sErrorDescription2 								:= UDINT_TO_STRING(udiHighLevelErrorId); 
			END_IF
			IF bLowLevelErrorRCActive THEN
				udiLowLevelErrorId								:= IODATA;
				//udiErrorId										:= 311;
				sErrorDescription2 								:= UDINT_TO_STRING(udiHighLevelErrorId); 
				//Opis błędu
			END_IF	
			
			ErrorDescription();
			arfbAlarm[0].ipArguments.Clear() .AddString(sErrorDescription1);
				
				IF NOT arfbAlarm[0].bActive THEN	
		 			arfbAlarm[0].Raise(nTimeStamp:=0);
		 		END_IF
				
				
		
		ELSIF bErrorNumberRequestActive  AND IODATA = 50 AND bEStop THEN
			
				sErrorDescription1								:= '';
				sErrorDescription2 								:= ''; 
				bError											:= FALSE;
				bResetErrorRC									:= TRUE;
		END_IF
	
	END_IF	
 	

// 	IF bErrorRCActive AND bLowLevelErrorRCActive AND NOT bStateError THEN
// 		
// 		bError											:= TRUE;
// 		bErrorNumberRequest								:= TRUE;
// 		udiLowLevelErrorId								:= IODATA;
// 		udiErrorId										:= 311;
// 		udiErrorId										:= udiLowLevelErrorId; 
	
ELSE
//	IF  arfbAlarm[0].bActive AND bReset THEN
//	//bServoONRC							:= FALSE;	
// 		arfbAlarm[0].Clear(nTimeStamp:=0, bResetConfirmation:= FALSE);
//	END_IF
	bErrorNumberRequest									:= FALSE;	
	bError												:= 	FALSE;
	sErrorDescription1									:= '';
	sErrorDescription2 									:= ''; 
		
END_IF

(*Wyświetlanie błedu na wyjściu*)
bError							:= FALSE;
FOR nAlarmNumerator := 0 TO 19 DO
	bError						:= bError OR arfbAlarm[nAlarmNumerator].bActive;
END_FOR
	

// Przejście do eError
IF (bError AND NOT bStateError AND bEStop) THEN
	eState												:= 	E_Station.eError;
END_IF

sErrorStationName 					:= sStationName;
END_ACTION

ACTION Homing:
CASE iCaseHoming OF
	0:
		iCaseRC							:= 100;
		iCaseInit						:=0;
		IF iActualCase = 100 THEN
			iCaseRC						:= 0;
			iCaseHoming					:= 10;
		END_IF
	10:
		IF iActualCase = 150 THEN
			eState						:= E_Station.eHomingDone;
			bHomingDone					:= TRUE;
		END_IF	
END_CASE
END_ACTION

ACTION Init:
tonRetryInit(IN:=(iCaseInit = 20 OR iCaseInit = 30 OR iCaseInit = 60), PT:=T#5S);
tonReadyError(IN:=(iCaseInit=0), PT:=T#30S);

CASE iCaseInit OF
	0:
		iCaseRC								:= 0;
		bOperationEnableRC					:= FALSE;
		bServoONRC							:= FALSE;
		bRunProgramRC						:= FALSE;
		bProgramResetRC						:= FALSE;
		IF bReadyRC THEN            		
			iCaseInit						:= 10;
		END_IF                      		
	10:		                        	
		bOperationEnableRC 					:= TRUE;
		IF bOperationEnableRCActive THEN
			iCaseInit						:= 30;			//25.09.2020
		END_IF
	20:
		bProgramResetRC						:= TRUE;
		IF bProgramSelectRCActive THEN
			bProgramResetRC					:= FALSE;
			iCaseInit						:= 30;
		END_IF
		IF tonRetryInit.Q THEN
			iCaseInit						:= 0;
		END_IF
		
	30: // Reset bledu od estopa
	
		bErrorNumberRequest					:= TRUE;
		
		IF bErrorNumberRequestActive  THEN
			udiErrorIdInit					:= IODATA;	
			iCaseInit						:= iCaseInit + 10;	
		END_IF
	40: //	
		IF 	udiErrorIdInit = 50 THEN
			bResetErrorRC					:= TRUE;
			bErrorNumberRequest				:= FALSE;
			iCaseInit						:= iCaseInit +10;			
		ELSE
				iCaseInit					:= 60;
		END_IF
		
	50://
		IF 	NOT bErrorRCActive THEN
			bResetErrorRC					:= FALSE;
			iCaseInit						:= iCaseInit +10;
		END_IF		
				
	60:
		bServoONRC							:= TRUE;
		IF bServoONRCActive THEN
			iCaseInit						:= 70;
		END_IF
		IF tonRetryInit.Q THEN
			iCaseInit						:= 0;
		END_IF
	70:
		bRunProgramRC						:= TRUE;
		IF bRunProgramRCActive THEN
			iCaseInit						:= 80;
		END_IF
						
	80:
		eState 				 				:= E_Station.eReady;
	
END_CASE
END_ACTION

ACTION LubricationCounter:
(*Zliczanie cykli robota*)
rtPick(CLK:=bRun, Q=>);
IF rtPick.Q THEN
	nLubricationCounter := nLubricationCounter + 1;
END_IF
END_ACTION

ACTION Maintenance:
// Trzeba zmienic ta nazwe na wymiane baterii
IF bBatteryReplacementWasMade  THEN
	
	bBatteryReplacementDone						:= TRUE;
ELSE             
                           	
	bBatteryReplacementDone						:= FALSE;	
	
END_IF

// Wymiana Smaru

IF bGreaseReplacementWasMade AND iAxisId =1 THEN
	
	bOperationEnableRC							:= TRUE;	
	bGreaseReplacementDoneAxis1					:= TRUE;

	
ELSIF bGreaseReplacementWasMade AND iAxisId =2 THEN
	
	bOperationEnableRC							:= TRUE;
	bGreaseReplacementDoneAxis2					:= TRUE;
		
	
ELSIF bGreaseReplacementWasMade AND iAxisId =3 THEN
	
	bOperationEnableRC							:= TRUE;		
	bGreaseReplacementDoneAxis3					:= TRUE;
	
ELSE
	
	bGreaseReplacementDoneAxis1					:= FALSE;	
	bGreaseReplacementDoneAxis2					:= FALSE;
	bGreaseReplacementDoneAxis3					:= FALSE;	
	
END_IF


// Wymiana paska
IF bBeltReplacementWasMade AND iAxisId = 3 THEN
	
	bOperationEnableRC							:= TRUE;		
	bBeltReplacementDoneAxis3					:= TRUE;
	
ELSIF bBeltReplacementWasMade AND iAxisId = 4 THEN
	
	bOperationEnableRC							:= TRUE;		
	bBeltReplacementDoneAxis4					:= TRUE;
	
ELSE
	
	bBeltReplacementDoneAxis3					:= FALSE;	
	bBeltReplacementDoneAxis4					:= FALSE;

END_IF


// Reset wymiany smaru 
IF bGreaseReplacementDoneAxis1 THEN
	
	bGreaseReplacementDone 						:= TRUE;
	udiIoDATARCWrite							:= 2;
	
ELSIF bGreaseReplacementDoneAxis2 THEN	
	
	bGreaseReplacementDone 						:= TRUE;
	udiIoDATARCWrite							:= 2;

ELSIF bGreaseReplacementDoneAxis3 THEN	
	
	bGreaseReplacementDone 						:= TRUE;
	udiIoDATARCWrite							:= 4;	

ELSE
	
	bGreaseReplacementDone 						:= FALSE;	
	
END_IF

// Reset wymiany paska
IF bBeltReplacementDoneAxis3 THEN
	
	bBeltReplacementDone 						:= TRUE;
	udiIoDATARCWrite							:= 4;
	
ELSIF bBeltReplacementDoneAxis4 THEN
	
	bBeltReplacementDone 						:= TRUE;
	udiIoDATARCWrite							:= 8;	
	
ELSE
	
	bBeltReplacementDone 						:= FALSE;	
	
END_IF


// Zerowanie rozkazu resetu
IF bBatteryReplenishmentFinished THEN
	
	bBatteryReplacementDone						:= FALSE;	
	bBatteryReplacementWasMade 					:= FALSE;	
	
END_IF

IF bGreaseReplenishmentFinished THEN
	
	bGreaseReplacementDone 						:= FALSE;	
	bGreaseReplacementWasMade					:= FALSE;
	
END_IF

IF bBeltReplenishmentFinished THEN
	
	bBeltReplacementDone 						:= FALSE;
	bBeltReplacementWasMade						:= FALSE;	
	
END_IF


// Wyzerowanie wartości wpisywanej do robota
IF NOT bGreaseReplacementDoneAxis1 AND NOT bGreaseReplacementDoneAxis2 AND NOT bGreaseReplacementDoneAxis3 AND NOT bBeltReplacementDoneAxis3 AND NOT bBeltReplacementDoneAxis4 THEN
	udiIoDATARCWrite							:= 0;	
END_IF
END_ACTION

ACTION ManualMovements:
// Zboacze narastajace aktywacji edytowania ofsetu
ftCapFeederRobotEditOffset(CLK:=bEditOffset);
// Zboacze opadajace aktywacji edytowania ofsetu
rtCapFeederRobotEditOffset(CLK:=bEditOffset);

//Wywoluje akcje Maintenence do resetowania czasow baterii, smarowania i wymiany paska

Maintenance();


IF ftCapFeederRobotEditOffset.Q THEN
	bComingUp											:= TRUE;
	iCaseRC												:= 0;	
	
	//? VIS.bCapFeederRobotManualPickPlace1					:= FALSE;
	//?  VIS.bCapFeederRobotManualPickPlace2					:= FALSE;
	//?  VIS.bCapFeederRobotManualPlace						:= FALSE;
	
END_IF
IF rtCapFeederRobotEditOffset.Q THEN
	bComingUp											:= TRUE;
	bManualCatch										:= NOT bCatcherCloseSensor;
END_IF


